// TIA Portal V19 program export: 2 tag tables, 1 data types, 4 data blocks, 27 code blocks (in call order from the OBs), 31 instance data blocks

VAR_GLOBAL   // PLC tag table "Default tag table"
   B0 AT %QB0 : Byte;
   B1 AT %QB1 : Byte;
   Clock_Byte AT %MB0 : Byte;
   Clock_10Hz AT %M0.0 : Bool;
   Clock_5Hz AT %M0.1 : Bool;
   "Clock_2.5Hz" AT %M0.2 : Bool;
   Clock_2Hz AT %M0.3 : Bool;
   "Clock_1.25Hz" AT %M0.4 : Bool;
   Clock_1Hz AT %M0.5 : Bool;
   "Clock_0.625Hz" AT %M0.6 : Bool;
   "Clock_0.5Hz" AT %M0.7 : Bool;
   System_Byte AT %MB1 : Byte;
   FirstScan AT %M1.0 : Bool;
   DiagStatusUpdate AT %M1.1 : Bool;
   AlwaysTRUE AT %M1.2 : Bool;
   AlwaysFALSE AT %M1.3 : Bool;
   "from et200sp PLC_1" AT %IB100 : Byte;   // Clock Byte From ET200SP sent Left Coupler for Display on RIO 1
   toET200spfromPLC1 AT %QB100 : Byte;   // Clock Byte To ET200SP sent Left Coupler
   "from et200sp PLC_1 Right" AT %IB200 : Byte;   // Clock Byte From ET200SP sent Right Coupler for Display on RIO 1
   "toET200spfromPLC1 Right" AT %QB200 : Byte;   // Clock Byte To ET200SP sent Right Coupler
END_VAR

VAR_GLOBAL   // PLC tag table "LAcycCom_Common"
END_VAR
VAR_GLOBAL CONSTANT   // user constants
   LACYCCOM_BUFFER_ELEMENTS_UPPER_LIM : Int := 59;   // Upper limit of request buffer array
END_VAR

TYPE "NetworkSwitchHMI"
   STRUCT
      Ports { S7_SetPoint := 'True'} : Array[1..8] of "LPNDR_typePortInformation";
      Port { S7_SetPoint := 'True'} : "LPNDR_typePortInformation";
      Index { S7_SetPoint := 'True'} : Int := 1;
   END_STRUCT;
END_TYPE

DATA_BLOCK "GlobalDB"   // DB9
{ S7_Optimized_Access := 'FALSE' }
   VAR RETAIN
      RTInfo : Struct   // Used to collect runtime information on an individual FB/FC
         Mode : UInt := 1;
         OBnumber : OB_ANY := 1;
         Info_LTIME : LTime := LT#0NS;
         RetVal : Int := 0;
      END_STRUCT;
      Runtime : Struct   // Used to collect individual runtime information of OB
         OB1Scan : Struct
            Min : LReal := 1000.0;
            Max : LReal;
            Current { ExternalAccessible := 'False'; ExternalVisible := 'False'; ExternalWritable := 'False'} : LReal;
            temp { ExternalAccessible := 'False'; ExternalVisible := 'False'; ExternalWritable := 'False'} : LReal;
            Mem { ExternalAccessible := 'False'; ExternalVisible := 'False'; ExternalWritable := 'False'} : LReal := 0.0;
            PreviousScan { ExternalAccessible := 'False'; ExternalVisible := 'False'; ExternalWritable := 'False'} : LReal;
            ResetMin : Bool;
            "Reset Max" : Bool;
         END_STRUCT;
      END_STRUCT;
      Trigger_StopSynch : Struct   // Used to trigger the Swapping of Status on the Reundant PLC
         REQ_FullSwapSequence { S7_SetPoint := 'True'} : Bool;   // Trigger used to perform a full swap of PLCs
         REQ_StopPrimary { S7_SetPoint := 'True'} : Bool;   // trigger a primary stop
         REQ_SynchUp { S7_SetPoint := 'True'} : Bool;   // trigger a synchronization
         Mode_StopPrimary : Int := 8;   // Stop Primary = 8
         Mode_SynchUp : Int := 7;   // Synchronization = 7
         StopPrimary_Retry_Busy : Bool;   // triggered due to RHCTRL being busy
         SynchUp_Retry_Busy : Bool;   // triggered due to RHCTRL being busy
         SyncSequenceFlag : Bool;
         RH_CTRL_PrimaryStop : Struct   // Used to stop and synch primary or backup
            REQ : Bool;
            Ret_Val : Byte;
            Busy : Bool;
         END_STRUCT;
         RH_CTRL_SyncUp : Struct   // Used to stop and synch primary or backup
            REQ : Bool;
            Ret_Val : Byte;
            Busy : Bool;
         END_STRUCT;
         SyncSequenceTimer : IEC_TIMER;
         SequenceTimer : IEC_TIMER;   // Timer to sequence between stop and synch
         SequenceAlarm { S7_SetPoint := 'True'} : Bool;
      END_STRUCT;
      Network { S7_SetPoint := 'True'} : "NetworkSwitchHMI";   // Used to collect switch XC208 details
      SystemTime { S7_SetPoint := 'True'} : DTL;   // Used to record cycle time of code
      tempSystemTime { S7_SetPoint := 'True'} : Int;
      "Array" : Array[0..1000] of "typeDiagnostics";   // Test Array
   END_VAR
BEGIN
   Trigger_StopSynch.SequenceTimer.PT := T#25s;   // Time based on full sequence elapsed timer
END_DATA_BLOCK

DATA_BLOCK "DB_HMI Support"   // DB10000
{ S7_Optimized_Access := 'FALSE' }
// stored: AutoNumber false
   VAR
      "PLC Mode" : Int;
      "PLC Near Status" : Int;
      "PLC Far Status" : Int;
      "Bypasses Status" : Int;
      OperationStateSystem : Int;
      MRPRingState : Int;
   END_VAR
BEGIN
END_DATA_BLOCK

DATA_BLOCK "hmiDatatransferTP1200"   // DB10
{ S7_Optimized_Access := 'TRUE' }
// stored: AutoNumber false, MemoryReserve 100
   VAR
      plc1LedState : Int;
      plc2LedState : Int;
      plcOperationState : Int;
      plcMrpState : Int;
      plcStopMonitoring : Int;
   END_VAR
BEGIN
END_DATA_BLOCK

DATA_BLOCK "EnS_Buffer32469"   // DB2
TITLE = Global DB for buffer data
AUTHOR : Siemens
FAMILY : EnS
// Global DB for buffer data
   STRUCT
      EnS_Buffer32469 : Array[0..114] of "EnS_typeValue";
   END_STRUCT;
BEGIN
END_DATA_BLOCK

ORGANIZATION_BLOCK "Main"   // OB1, LAD, ProgramCycle
TITLE = "Main Program Sweep (Cycle)"
{ S7_Optimized_Access := 'TRUE' }
// stored: AutoNumber false, SetENOAutomatically false
   VAR_INPUT
      Initial_Call : Bool;   // Initial call of this OB
      Remanence : Bool;   // =True, if remanent data are available
   END_VAR
BEGIN

REGION Network 1: Map clock byte to output of dq card
   // Display "to" and "from" using move command for troubleshooting
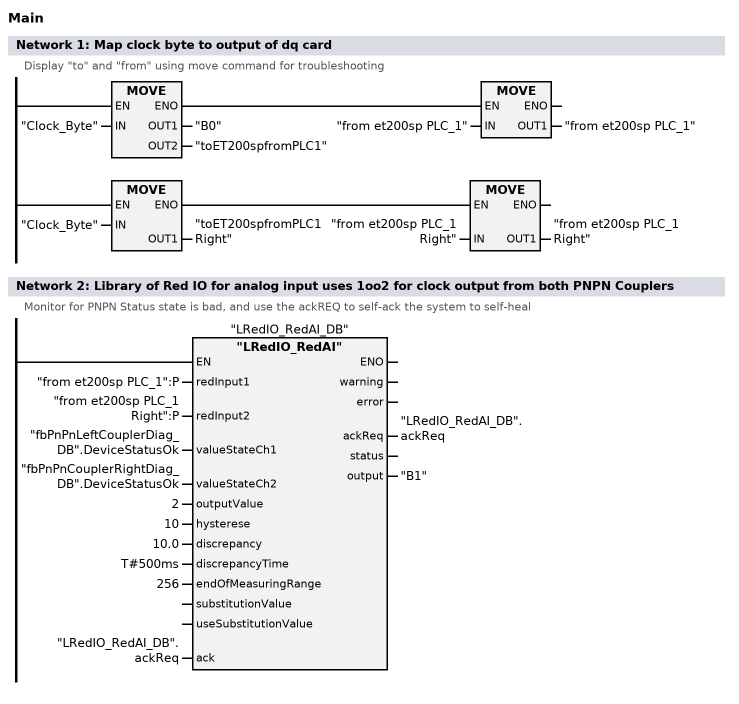
   RUNG wire#powerrail
      Move(in := "Clock_Byte", out1 => "B0", out2 => "toET200spfromPLC1")
      Move(in := "from et200sp PLC_1", out1 => "from et200sp PLC_1")
   END_RUNG
   RUNG wire#powerrail
      Move(in := "Clock_Byte", out1 => "toET200spfromPLC1 Right")
      Move(in := "from et200sp PLC_1 Right", out1 => "from et200sp PLC_1 Right")
   END_RUNG
   // the same network as SCL:
   "B0" := "Clock_Byte";
   "toET200spfromPLC1" := "Clock_Byte";
   "from et200sp PLC_1" := "from et200sp PLC_1";
   "toET200spfromPLC1 Right" := "Clock_Byte";
   "from et200sp PLC_1 Right" := "from et200sp PLC_1 Right";
END_REGION

REGION Network 2: Library of Red IO for analog input uses 1oo2 for clock output from both PNPN Couplers
   // Monitor for PNPN Status state is bad, and use the ackREQ to self-ack the system to self-heal
   RUNG wire#powerrail
      "LRedIO_RedAI_DB"(redInput1 := "from et200sp PLC_1":P, redInput2 := "from et200sp PLC_1 Right":P, valueStateCh1 := "fbPnPnLeftCouplerDiag_DB".DeviceStatusOk, valueStateCh2 := "fbPnPnCouplerRightDiag_DB".DeviceStatusOk, outputValue := 2, hysterese := 10, discrepancy := 10.0, discrepancyTime := T#500ms, endOfMeasuringRange := 256, substitutionValue :=, useSubstitutionValue :=, ack := "LRedIO_RedAI_DB".ackReq, warning =>, error =>, ackReq => "LRedIO_RedAI_DB".ackReq, status =>, output => "B1")
   END_RUNG
   // the same network as SCL:
   "LRedIO_RedAI_DB"(redInput1 := "from et200sp PLC_1":P,   // "LRedIO_RedAI"
                     redInput2 := "from et200sp PLC_1 Right":P,
                     valueStateCh1 := "fbPnPnLeftCouplerDiag_DB".DeviceStatusOk,
                     valueStateCh2 := "fbPnPnCouplerRightDiag_DB".DeviceStatusOk,
                     outputValue := 2,
                     hysterese := 10,
                     discrepancy := 10.0,
                     discrepancyTime := T#500ms,
                     endOfMeasuringRange := 256,
                     ack := "LRedIO_RedAI_DB".ackReq,
                     ackReq => "LRedIO_RedAI_DB".ackReq,
                     output => "B1");
END_REGION
END_ORGANIZATION_BLOCK

ORGANIZATION_BLOCK "RT_Info_Cyclic"   // OB30, LAD, CyclicInterrupt
{ S7_Optimized_Access := 'TRUE' }
// stored: SetENOAutomatically false
   VAR_INPUT
      Initial_Call : Bool;   // Initial call of this OB
      Event_Count : Int;   // Events discarded
   END_VAR
   VAR CONSTANT
      constRunSoloState : Int := 37;
      constRunRedundant : Int := 40;
   END_VAR
   VAR_TEMP   // added for the SCL form of the ladder/FBD networks
      _w1 : Bool;
      _w2 : Bool;
      _w3 : Bool;
      _w4 : Bool;
   END_VAR
BEGIN

REGION Network 1: RT_Info for specific OB
   // Used to find the specific runtime of an OB, change the OB number and see the INFO.
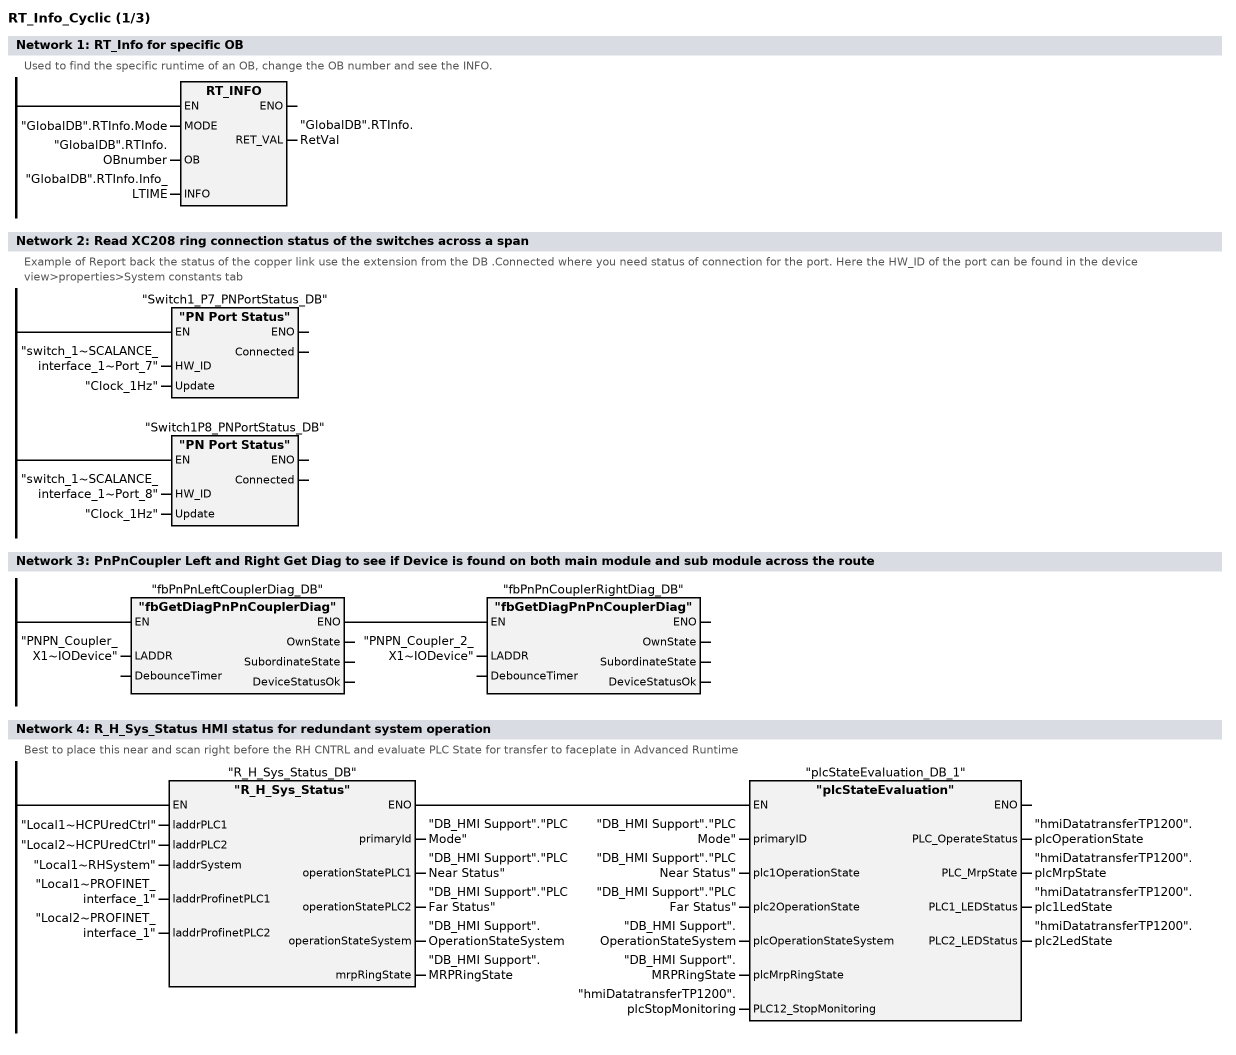
   RUNG wire#powerrail
      RT_INFO(MODE := "GlobalDB".RTInfo.Mode, OB := "GlobalDB".RTInfo.OBnumber, INFO := "GlobalDB".RTInfo.Info_LTIME, Ret_Val => "GlobalDB".RTInfo.RetVal)
   END_RUNG
   // the same network as SCL:
   "GlobalDB".RTInfo.RetVal := RT_INFO(MODE := "GlobalDB".RTInfo.Mode,
                           OB := "GlobalDB".RTInfo.OBnumber,
                           INFO := "GlobalDB".RTInfo.Info_LTIME);
END_REGION

REGION Network 2: Read XC208 ring connection status of the switches across a span
   // Example of Report back the status of the copper link use the extension from the DB .Connected where you need status of connection for the port. Here the HW_ID of the port can be found in the device view>properties>System constants tab
   RUNG wire#powerrail
      "Switch1_P7_PNPortStatus_DB"(HW_ID := "switch_1~SCALANCE_interface_1~Port_7", Update := "Clock_1Hz", Connected =>)
   END_RUNG
   RUNG wire#powerrail
      "Switch1P8_PNPortStatus_DB"(HW_ID := "switch_1~SCALANCE_interface_1~Port_8", Update := "Clock_1Hz", Connected =>)
   END_RUNG
   // the same network as SCL:
   "Switch1_P7_PNPortStatus_DB"(HW_ID := "switch_1~SCALANCE_interface_1~Port_7", Update := "Clock_1Hz");   // "PN Port Status"
   "Switch1P8_PNPortStatus_DB"(HW_ID := "switch_1~SCALANCE_interface_1~Port_8", Update := "Clock_1Hz");   // "PN Port Status"
END_REGION

REGION Network 3: PnPnCoupler Left and Right Get Diag to see if Device is found on both main module and sub module across the route
   RUNG wire#powerrail
      "fbPnPnLeftCouplerDiag_DB"(LADDR := "PNPN_Coupler_X1~IODevice", DebounceTimer :=, OwnState =>, SubordinateState =>, DeviceStatusOk =>)
      "fbPnPnCouplerRightDiag_DB"(LADDR := "PNPN_Coupler_2_X1~IODevice", DebounceTimer :=, OwnState =>, SubordinateState =>, DeviceStatusOk =>)
   END_RUNG
   // the same network as SCL:
   "fbPnPnLeftCouplerDiag_DB"(LADDR := "PNPN_Coupler_X1~IODevice", ENO => #_w1);   // "fbGetDiagPnPnCouplerDiag"
   IF #_w1 THEN
       "fbPnPnCouplerRightDiag_DB"(LADDR := "PNPN_Coupler_2_X1~IODevice");   // "fbGetDiagPnPnCouplerDiag"
   END_IF;
END_REGION

REGION Network 4: R_H_Sys_Status HMI status for redundant system operation
   // Best to place this near and scan right before the RH CNTRL and evaluate PLC State for transfer to faceplate in Advanced Runtime
   RUNG wire#powerrail
      "R_H_Sys_Status_DB"(laddrPLC1 := "Local1~HCPUredCtrl", laddrPLC2 := "Local2~HCPUredCtrl", laddrSystem := "Local1~RHSystem", laddrProfinetPLC1 := "Local1~PROFINET_interface_1", laddrProfinetPLC2 := "Local2~PROFINET_interface_1", primaryId => "DB_HMI Support"."PLC Mode", operationStatePLC1 => "DB_HMI Support"."PLC Near Status", operationStatePLC2 => "DB_HMI Support"."PLC Far Status", operationStateSystem => "DB_HMI Support".OperationStateSystem, mrpRingState => "DB_HMI Support".MRPRingState)
      "plcStateEvaluation_DB_1"(primaryID := "DB_HMI Support"."PLC Mode", plc1OperationState := "DB_HMI Support"."PLC Near Status", plc2OperationState := "DB_HMI Support"."PLC Far Status", plcOperationStateSystem := "DB_HMI Support".OperationStateSystem, plcMrpRingState := "DB_HMI Support".MRPRingState, PLC12_StopMonitoring := "hmiDatatransferTP1200".plcStopMonitoring, PLC_OperateStatus => "hmiDatatransferTP1200".plcOperationState, PLC_MrpState => "hmiDatatransferTP1200".plcMrpState, PLC1_LEDStatus => "hmiDatatransferTP1200".plc1LedState, PLC2_LEDStatus => "hmiDatatransferTP1200".plc2LedState)
   END_RUNG
   // the same network as SCL:
   "R_H_Sys_Status_DB"(laddrPLC1 := "Local1~HCPUredCtrl",   // "R_H_Sys_Status"
                       laddrPLC2 := "Local2~HCPUredCtrl",
                       laddrSystem := "Local1~RHSystem",
                       laddrProfinetPLC1 := "Local1~PROFINET_interface_1",
                       laddrProfinetPLC2 := "Local2~PROFINET_interface_1",
                       primaryId => "DB_HMI Support"."PLC Mode",
                       operationStatePLC1 => "DB_HMI Support"."PLC Near Status",
                       operationStatePLC2 => "DB_HMI Support"."PLC Far Status",
                       operationStateSystem => "DB_HMI Support".OperationStateSystem,
                       mrpRingState => "DB_HMI Support".MRPRingState,
                       ENO => #_w1);
   IF #_w1 THEN
       "plcStateEvaluation_DB_1"(primaryID := "DB_HMI Support"."PLC Mode",   // "plcStateEvaluation"
                               plc1OperationState := "DB_HMI Support"."PLC Near Status",
                               plc2OperationState := "DB_HMI Support"."PLC Far Status",
                               plcOperationStateSystem := "DB_HMI Support".OperationStateSystem,
                               plcMrpRingState := "DB_HMI Support".MRPRingState,
                               PLC12_StopMonitoring := "hmiDatatransferTP1200".plcStopMonitoring,
                               PLC_OperateStatus => "hmiDatatransferTP1200".plcOperationState,
                               PLC_MrpState => "hmiDatatransferTP1200".plcMrpState,
                               PLC1_LEDStatus => "hmiDatatransferTP1200".plc1LedState,
                               PLC2_LEDStatus => "hmiDatatransferTP1200".plc2LedState);
   END_IF;
END_REGION

REGION Network 5: Trigger primary stop RH_CNTRL
   // Self Latching Sequence using FullSwap Sequence tag, independent function with REQ tag
   // Used to trigger Primary Stop based on input from stop primary and full swap boolean tag;
   //  positive edge triggered instruction RH_CTRL below.
   // This network uses a Primary stop request, and evaluates if the RH_CTRL is busy before 
   // changing the mode or moving on to the next step.
   // The Retry_Busy tag is used to record if a Busy bit was in place while being triggered to prevent moving
   //  mode during middle of RH_CTRL operation.
   // 
   // Modes:
   // 3: Disable execution of the SYNCUP
   // 4: Re-enable execution of the SYNCUP
   // 7: Request SYNCUP system state 
   // 8: Request STOP of the primary CPU
   // 9: Request STOP of the backup CPU
   // 
   // Use mode 8 to stop the primary PLC, then use Mode 7 to Synch the primary and backup.
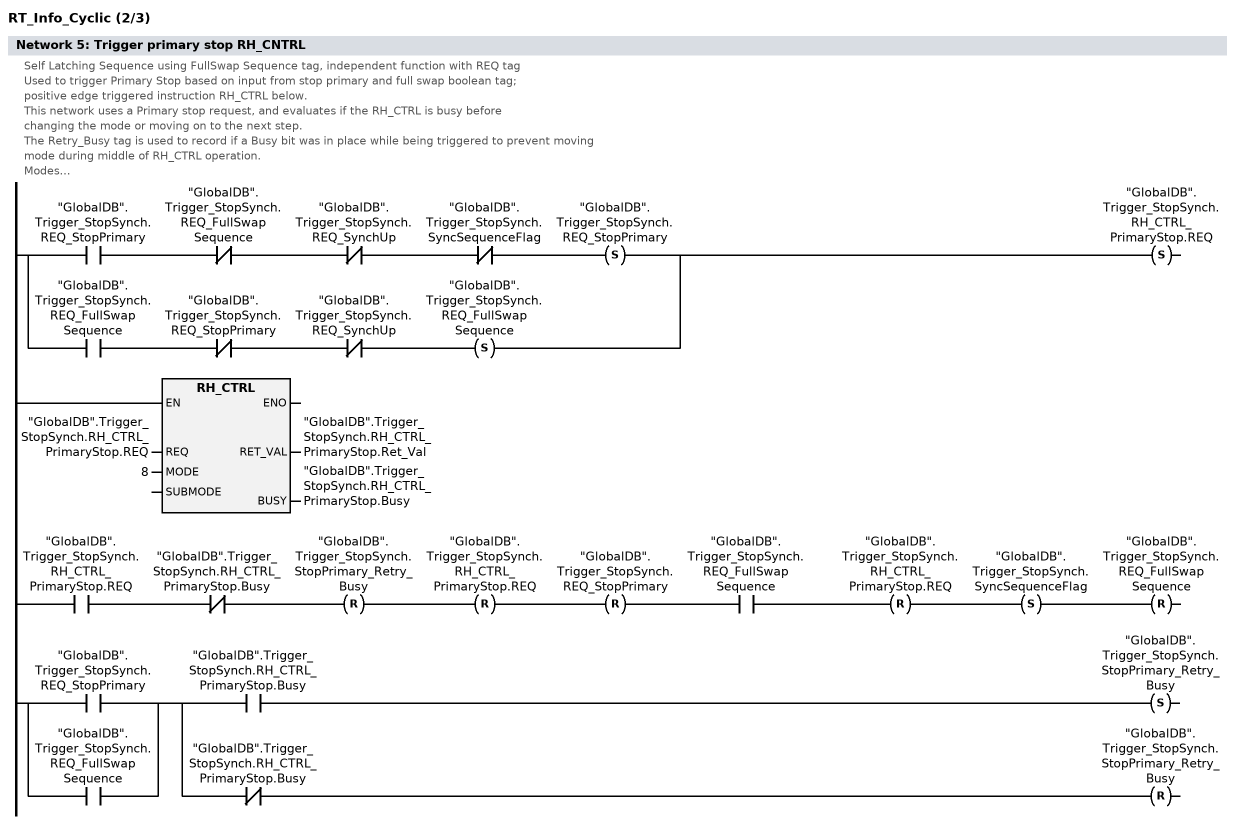
   RUNG wire#powerrail
      Contact( "GlobalDB".Trigger_StopSynch.REQ_StopPrimary )
      I_Contact( "GlobalDB".Trigger_StopSynch.REQ_FullSwapSequence )
      I_Contact( "GlobalDB".Trigger_StopSynch.REQ_SynchUp )
      I_Contact( "GlobalDB".Trigger_StopSynch.SyncSequenceFlag )
      S_Coil( "GlobalDB".Trigger_StopSynch.REQ_StopPrimary )
      wire#w1
      S_Coil( "GlobalDB".Trigger_StopSynch.RH_CTRL_PrimaryStop.REQ )
   END_RUNG
   RUNG wire#powerrail
      Contact( "GlobalDB".Trigger_StopSynch.REQ_FullSwapSequence )
      I_Contact( "GlobalDB".Trigger_StopSynch.REQ_StopPrimary )
      I_Contact( "GlobalDB".Trigger_StopSynch.REQ_SynchUp )
      S_Coil( "GlobalDB".Trigger_StopSynch.REQ_FullSwapSequence )
   END_RUNG wire#w1
   RUNG wire#powerrail
      RH_CTRL(REQ := "GlobalDB".Trigger_StopSynch.RH_CTRL_PrimaryStop.REQ, Mode := 8, Submode :=, Ret_Val => "GlobalDB".Trigger_StopSynch.RH_CTRL_PrimaryStop.Ret_Val, Busy => "GlobalDB".Trigger_StopSynch.RH_CTRL_PrimaryStop.Busy)
   END_RUNG
   RUNG wire#powerrail
      Contact( "GlobalDB".Trigger_StopSynch.RH_CTRL_PrimaryStop.REQ )
      I_Contact( "GlobalDB".Trigger_StopSynch.RH_CTRL_PrimaryStop.Busy )
      R_Coil( "GlobalDB".Trigger_StopSynch.StopPrimary_Retry_Busy )
      R_Coil( "GlobalDB".Trigger_StopSynch.RH_CTRL_PrimaryStop.REQ )
      R_Coil( "GlobalDB".Trigger_StopSynch.REQ_StopPrimary )
      Contact( "GlobalDB".Trigger_StopSynch.REQ_FullSwapSequence )
      R_Coil( "GlobalDB".Trigger_StopSynch.RH_CTRL_PrimaryStop.REQ )
      S_Coil( "GlobalDB".Trigger_StopSynch.SyncSequenceFlag )
      R_Coil( "GlobalDB".Trigger_StopSynch.REQ_FullSwapSequence )
   END_RUNG
   RUNG wire#powerrail
      Contact( "GlobalDB".Trigger_StopSynch.REQ_StopPrimary )
      wire#w2
      Contact( "GlobalDB".Trigger_StopSynch.RH_CTRL_PrimaryStop.Busy )
      S_Coil( "GlobalDB".Trigger_StopSynch.StopPrimary_Retry_Busy )
   END_RUNG
   RUNG wire#powerrail
      Contact( "GlobalDB".Trigger_StopSynch.REQ_FullSwapSequence )
   END_RUNG wire#w2
   RUNG wire#w2
      I_Contact( "GlobalDB".Trigger_StopSynch.RH_CTRL_PrimaryStop.Busy )
      R_Coil( "GlobalDB".Trigger_StopSynch.StopPrimary_Retry_Busy )
   END_RUNG
   // the same network as SCL:
   #_w1 := "GlobalDB".Trigger_StopSynch.REQ_StopPrimary AND NOT "GlobalDB".Trigger_StopSynch.REQ_FullSwapSequence AND NOT "GlobalDB".Trigger_StopSynch.REQ_SynchUp AND NOT "GlobalDB".Trigger_StopSynch.SyncSequenceFlag;
   IF #_w1 THEN "GlobalDB".Trigger_StopSynch.REQ_StopPrimary := TRUE; END_IF;
   #_w2 := "GlobalDB".Trigger_StopSynch.REQ_FullSwapSequence AND NOT "GlobalDB".Trigger_StopSynch.REQ_StopPrimary AND NOT "GlobalDB".Trigger_StopSynch.REQ_SynchUp;
   IF #_w2 THEN "GlobalDB".Trigger_StopSynch.REQ_FullSwapSequence := TRUE; END_IF;
   IF #_w1 OR #_w2 THEN "GlobalDB".Trigger_StopSynch.RH_CTRL_PrimaryStop.REQ := TRUE; END_IF;
   "GlobalDB".Trigger_StopSynch.RH_CTRL_PrimaryStop.Ret_Val := RH_CTRL(REQ := "GlobalDB".Trigger_StopSynch.RH_CTRL_PrimaryStop.REQ,
                           Mode := 8,
                           Busy => "GlobalDB".Trigger_StopSynch.RH_CTRL_PrimaryStop.Busy);
   #_w3 := "GlobalDB".Trigger_StopSynch.RH_CTRL_PrimaryStop.REQ AND NOT "GlobalDB".Trigger_StopSynch.RH_CTRL_PrimaryStop.Busy;
   IF #_w3 THEN
       "GlobalDB".Trigger_StopSynch.StopPrimary_Retry_Busy := FALSE;
       "GlobalDB".Trigger_StopSynch.RH_CTRL_PrimaryStop.REQ := FALSE;
       "GlobalDB".Trigger_StopSynch.REQ_StopPrimary := FALSE;
   END_IF;
   IF #_w3 AND "GlobalDB".Trigger_StopSynch.REQ_FullSwapSequence THEN
       "GlobalDB".Trigger_StopSynch.RH_CTRL_PrimaryStop.REQ := FALSE;
       "GlobalDB".Trigger_StopSynch.SyncSequenceFlag := TRUE;
       "GlobalDB".Trigger_StopSynch.REQ_FullSwapSequence := FALSE;
   END_IF;
   #_w4 := "GlobalDB".Trigger_StopSynch.REQ_StopPrimary OR "GlobalDB".Trigger_StopSynch.REQ_FullSwapSequence;
   IF #_w4 AND "GlobalDB".Trigger_StopSynch.RH_CTRL_PrimaryStop.Busy THEN
       "GlobalDB".Trigger_StopSynch.StopPrimary_Retry_Busy := TRUE;
   END_IF;
   IF #_w4 AND NOT "GlobalDB".Trigger_StopSynch.RH_CTRL_PrimaryStop.Busy THEN
       "GlobalDB".Trigger_StopSynch.StopPrimary_Retry_Busy := FALSE;
   END_IF;
END_REGION

REGION Network 6: Trigger Synch up RH_CNTRL
   // Self Latching Sequence using FullSwap Sequence tag, independent function with REQ tag
   // Used to trigger Sync up; positive edge triggered instruction RH_CTRL below
   // Sequence can also be triggered by Full sequence request which can set the SyncSequenceFlag below
   // SyncSequence Flag is help for next step until run Run-Solo status is reported
   //  positive edge triggered instruction RH_CTRL below
   // This network uses a synch up request, and evaluates if the RH_CTRL is busy before changing the mode
   // The Retry_Busy tag is used to record if a Busy bit was in place while being triggered to prevent moving
   //  mode during middle of RH_CTRL operation
   // 
   // Modes:
   // 3: Disable execution of the SYNCUP
   // 4: Re-enable execution of the SYNCUP
   // 7: Request SYNCUP system state 
   // 8: Request STOP of the primary CPU
   // 9: Request STOP of the backup CPU
   // 
   // Use mode 8 to stop the primary PLC, then use Mode 7 to Synch the primary and backup.
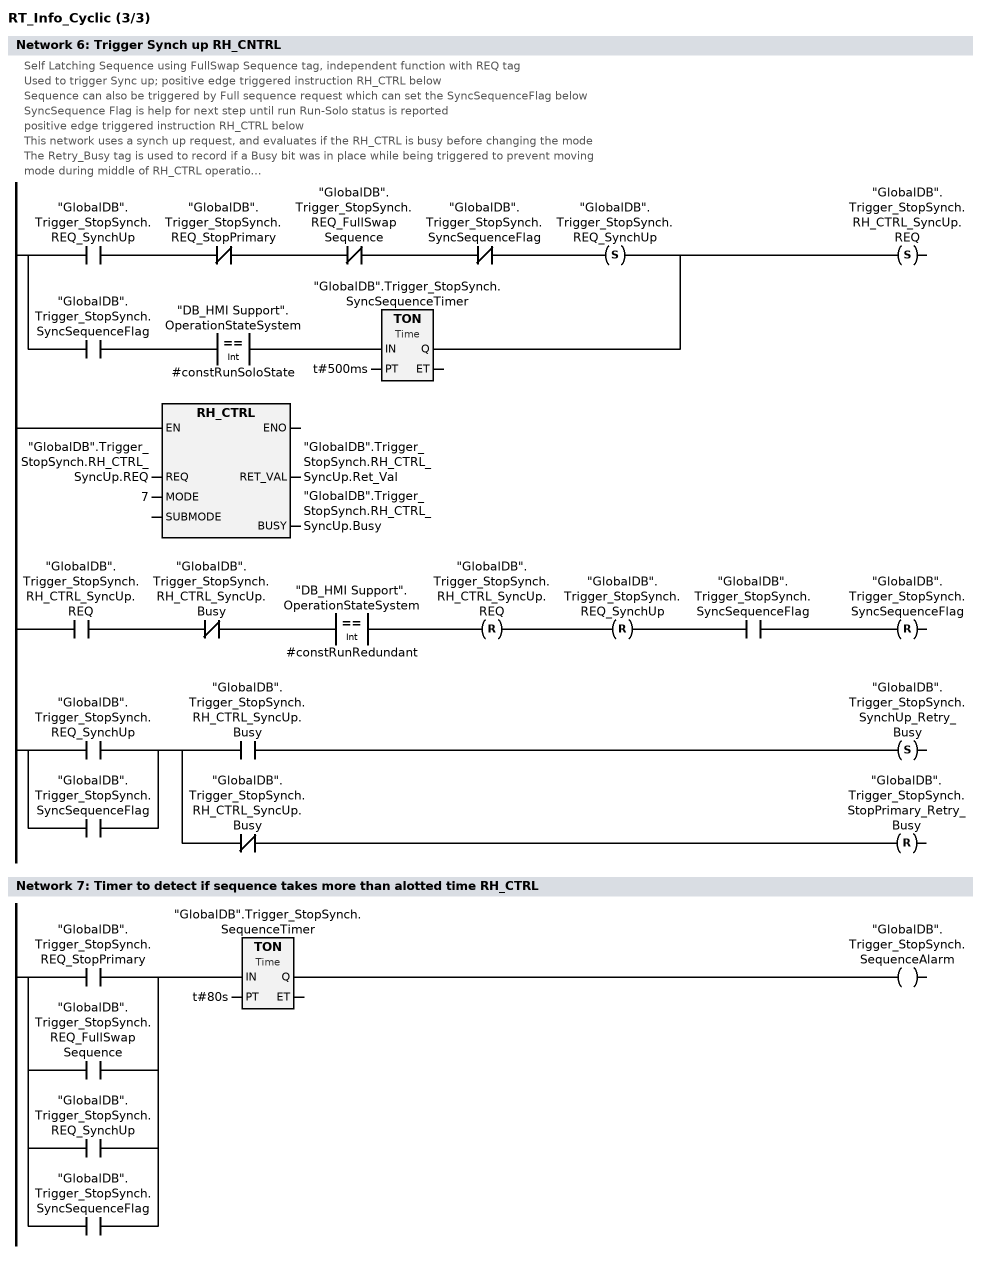
   RUNG wire#powerrail
      Contact( "GlobalDB".Trigger_StopSynch.REQ_SynchUp )
      I_Contact( "GlobalDB".Trigger_StopSynch.REQ_StopPrimary )
      I_Contact( "GlobalDB".Trigger_StopSynch.REQ_FullSwapSequence )
      I_Contact( "GlobalDB".Trigger_StopSynch.SyncSequenceFlag )
      S_Coil( "GlobalDB".Trigger_StopSynch.REQ_SynchUp )
      wire#w1
      S_Coil( "GlobalDB".Trigger_StopSynch.RH_CTRL_SyncUp.REQ )
   END_RUNG
   RUNG wire#powerrail
      Contact( "GlobalDB".Trigger_StopSynch.SyncSequenceFlag )
      { S7_Templates := "SrcType := Int" } EQ_Contact(in1 := "DB_HMI Support".OperationStateSystem, in2 := #constRunSoloState)
      { S7_Templates := "time_type := Time" } "GlobalDB".Trigger_StopSynch.SyncSequenceTimer.TON(pt := t#500ms, et =>)
   END_RUNG wire#w1
   RUNG wire#powerrail
      RH_CTRL(REQ := "GlobalDB".Trigger_StopSynch.RH_CTRL_SyncUp.REQ, Mode := 7, Submode :=, Ret_Val => "GlobalDB".Trigger_StopSynch.RH_CTRL_SyncUp.Ret_Val, Busy => "GlobalDB".Trigger_StopSynch.RH_CTRL_SyncUp.Busy)
   END_RUNG
   RUNG wire#powerrail
      Contact( "GlobalDB".Trigger_StopSynch.RH_CTRL_SyncUp.REQ )
      I_Contact( "GlobalDB".Trigger_StopSynch.RH_CTRL_SyncUp.Busy )
      { S7_Templates := "SrcType := Int" } EQ_Contact(in1 := "DB_HMI Support".OperationStateSystem, in2 := #constRunRedundant)
      R_Coil( "GlobalDB".Trigger_StopSynch.RH_CTRL_SyncUp.REQ )
      R_Coil( "GlobalDB".Trigger_StopSynch.REQ_SynchUp )
      Contact( "GlobalDB".Trigger_StopSynch.SyncSequenceFlag )
      R_Coil( "GlobalDB".Trigger_StopSynch.SyncSequenceFlag )
   END_RUNG
   RUNG wire#powerrail
      Contact( "GlobalDB".Trigger_StopSynch.REQ_SynchUp )
      wire#w2
      Contact( "GlobalDB".Trigger_StopSynch.RH_CTRL_SyncUp.Busy )
      S_Coil( "GlobalDB".Trigger_StopSynch.SynchUp_Retry_Busy )
   END_RUNG
   RUNG wire#powerrail
      Contact( "GlobalDB".Trigger_StopSynch.SyncSequenceFlag )
   END_RUNG wire#w2
   RUNG wire#w2
      I_Contact( "GlobalDB".Trigger_StopSynch.RH_CTRL_SyncUp.Busy )
      R_Coil( "GlobalDB".Trigger_StopSynch.StopPrimary_Retry_Busy )
   END_RUNG
   // the same network as SCL:
   #_w1 := "GlobalDB".Trigger_StopSynch.REQ_SynchUp AND NOT "GlobalDB".Trigger_StopSynch.REQ_StopPrimary AND NOT "GlobalDB".Trigger_StopSynch.REQ_FullSwapSequence AND NOT "GlobalDB".Trigger_StopSynch.SyncSequenceFlag;
   IF #_w1 THEN "GlobalDB".Trigger_StopSynch.REQ_SynchUp := TRUE; END_IF;
   "GlobalDB".Trigger_StopSynch.SyncSequenceTimer.TON(IN := "GlobalDB".Trigger_StopSynch.SyncSequenceFlag AND ("DB_HMI Support".OperationStateSystem = #constRunSoloState),
                           PT := t#500ms);
   IF #_w1 OR "GlobalDB".Trigger_StopSynch.SyncSequenceTimer.Q THEN
       "GlobalDB".Trigger_StopSynch.RH_CTRL_SyncUp.REQ := TRUE;
   END_IF;
   "GlobalDB".Trigger_StopSynch.RH_CTRL_SyncUp.Ret_Val := RH_CTRL(REQ := "GlobalDB".Trigger_StopSynch.RH_CTRL_SyncUp.REQ,
                           Mode := 7,
                           Busy => "GlobalDB".Trigger_StopSynch.RH_CTRL_SyncUp.Busy);
   #_w2 := "GlobalDB".Trigger_StopSynch.RH_CTRL_SyncUp.REQ AND NOT "GlobalDB".Trigger_StopSynch.RH_CTRL_SyncUp.Busy AND ("DB_HMI Support".OperationStateSystem = #constRunRedundant);
   IF #_w2 THEN
       "GlobalDB".Trigger_StopSynch.RH_CTRL_SyncUp.REQ := FALSE;
       "GlobalDB".Trigger_StopSynch.REQ_SynchUp := FALSE;
   END_IF;
   IF #_w2 AND "GlobalDB".Trigger_StopSynch.SyncSequenceFlag THEN
       "GlobalDB".Trigger_StopSynch.SyncSequenceFlag := FALSE;
   END_IF;
   #_w3 := "GlobalDB".Trigger_StopSynch.REQ_SynchUp OR "GlobalDB".Trigger_StopSynch.SyncSequenceFlag;
   IF #_w3 AND "GlobalDB".Trigger_StopSynch.RH_CTRL_SyncUp.Busy THEN
       "GlobalDB".Trigger_StopSynch.SynchUp_Retry_Busy := TRUE;
   END_IF;
   IF #_w3 AND NOT "GlobalDB".Trigger_StopSynch.RH_CTRL_SyncUp.Busy THEN
       "GlobalDB".Trigger_StopSynch.StopPrimary_Retry_Busy := FALSE;
   END_IF;
END_REGION

REGION Network 7: Timer to detect if sequence takes more than alotted time RH_CTRL
   RUNG wire#powerrail
      Contact( "GlobalDB".Trigger_StopSynch.REQ_StopPrimary )
      wire#w1
      { S7_Templates := "time_type := Time" } "GlobalDB".Trigger_StopSynch.SequenceTimer.TON(pt := t#80s, et =>)
      Coil( "GlobalDB".Trigger_StopSynch.SequenceAlarm )
   END_RUNG
   RUNG wire#powerrail
      Contact( "GlobalDB".Trigger_StopSynch.REQ_FullSwapSequence )
   END_RUNG wire#w1
   RUNG wire#powerrail
      Contact( "GlobalDB".Trigger_StopSynch.REQ_SynchUp )
   END_RUNG wire#w1
   RUNG wire#powerrail
      Contact( "GlobalDB".Trigger_StopSynch.SyncSequenceFlag )
   END_RUNG wire#w1
   // the same network as SCL:
   "GlobalDB".Trigger_StopSynch.SequenceTimer.TON(IN := "GlobalDB".Trigger_StopSynch.REQ_StopPrimary OR "GlobalDB".Trigger_StopSynch.REQ_FullSwapSequence OR "GlobalDB".Trigger_StopSynch.REQ_SynchUp OR "GlobalDB".Trigger_StopSynch.SyncSequenceFlag,
                           PT := t#80s);
   "GlobalDB".Trigger_StopSynch.SequenceAlarm := "GlobalDB".Trigger_StopSynch.SequenceTimer.Q;
END_REGION
END_ORGANIZATION_BLOCK

FUNCTION_BLOCK "PN Port Status"   // FB5, LAD
{ S7_Optimized_Access := 'TRUE' }
// stored: MemoryReserve 100, SetENOAutomatically false
   VAR_INPUT
      HW_ID : HW_IO;
      Update : Bool;
   END_VAR
   VAR_OUTPUT
      Connected : Bool;
   END_VAR
   VAR
      Updated_ReqP : Bool;
      Updated_Req : Bool;
      RDREC_Instance { S7_SetPoint := 'True'} : RDREC;
   END_VAR
   VAR_TEMP
      Record : Struct
         BlockType : Word;
         BlockLength : UInt;
         BlockVersionHigh : USInt;
         BlockVersionLow : USInt;
         Padding : Word;
         SlotNumber : Word;
         SubSlotNumber : Word;
         Data : Array[0..299] of Byte;
      END_STRUCT;
      n : Array[0..3] of UInt;
      LinkState : Word;
   END_VAR
   VAR_TEMP   // added for the SCL form of the ladder/FBD networks
      _w1 : Bool;
   END_VAR
BEGIN

REGION Network 1: Positive Edge triggered Update Req
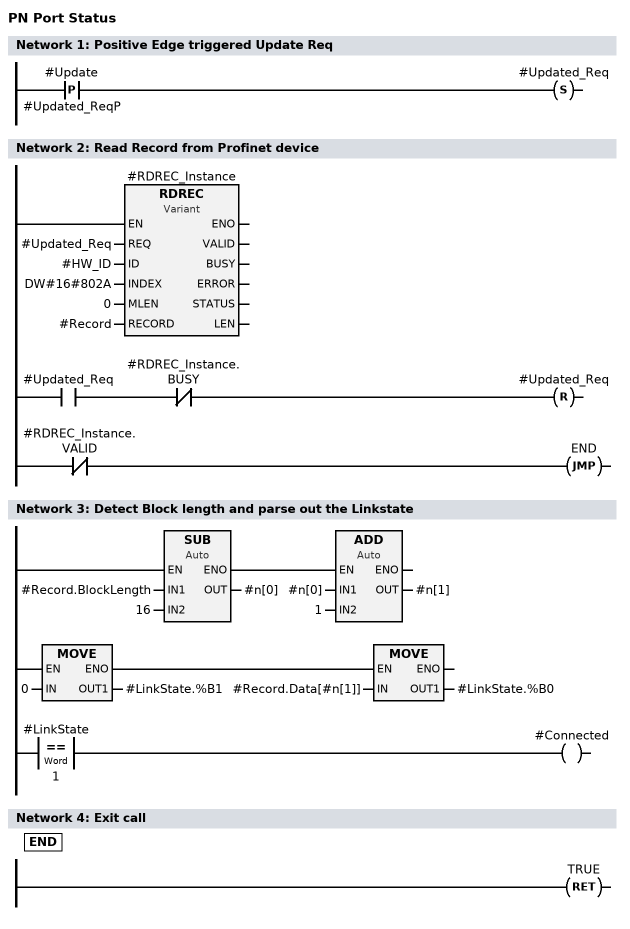
   RUNG wire#powerrail
      P_Contact(operand := #Update, bit := #Updated_ReqP)
      S_Coil( #Updated_Req )
   END_RUNG
   // the same network as SCL:
   #_w1 := #Update AND NOT #Updated_ReqP;   // rising edge of #Update
   #Updated_ReqP := #Update;
   IF #_w1 THEN #Updated_Req := TRUE; END_IF;
END_REGION

REGION Network 2: Read Record from Profinet device
   RUNG wire#powerrail
      { S7_Templates := "[ptr_type := Variant, id_type := HW_IO, index_type := DInt, len_type := UInt]" } #RDREC_Instance.RDREC(REQ := #Updated_Req, ID := #HW_ID, INDEX := DW#16#802A, MLEN := 0, RECORD := #Record, VALID =>, BUSY =>, ERROR =>, STATUS =>, LEN =>)
   END_RUNG
   RUNG wire#powerrail
      Contact( #Updated_Req )
      I_Contact( #RDREC_Instance.BUSY )
      R_Coil( #Updated_Req )
   END_RUNG
   RUNG wire#powerrail
      I_Contact( #RDREC_Instance.VALID )
      JumpCoil( END )
   END_RUNG
   // the same network as SCL:
   #RDREC_Instance(REQ := #Updated_Req, ID := #HW_ID, INDEX := DW#16#802A, MLEN := 0, RECORD := #Record);   // RDREC
   IF #Updated_Req AND NOT #RDREC_Instance.BUSY THEN #Updated_Req := FALSE; END_IF;
   IF NOT #RDREC_Instance.VALID THEN GOTO END; END_IF;
END_REGION

REGION Network 3: Detect Block length and parse out the Linkstate
   RUNG wire#powerrail
      Sub(in1 := #Record.BlockLength, in2 := 16, out => #n[0])
      Add(in1 := #n[0], in2 := 1, out => #n[1])
   END_RUNG
   RUNG wire#powerrail
      Move(in := 0, out1 => #LinkState.%B1)
      Move(in := #Record.Data[#n[1]], out1 => #LinkState.%B0)
   END_RUNG
   RUNG wire#powerrail
      { S7_Templates := "SrcType := Word" } EQ_Contact(in1 := #LinkState, in2 := 1)
      Coil( #Connected )
   END_RUNG
   // the same network as SCL:
   #n[0] := #Record.BlockLength - 16;
   #n[1] := #n[0] + 1;
   #LinkState.%B1 := 0;
   #LinkState.%B0 := #Record.Data[#n[1]];
   #Connected := #LinkState = 1;
END_REGION

REGION Network 4: Exit call
   END:
   ENO := TRUE;
   RETURN;
END_REGION
END_FUNCTION_BLOCK

FUNCTION_BLOCK "fbGetDiagPnPnCouplerDiag"   // FB1, LAD
{ S7_Optimized_Access := 'TRUE' }
// stored: MemoryReserve 100, SetENOAutomatically false
   VAR_INPUT
      LADDR : HW_ANY;   // Hardware Address of the ~IODevice number
      DebounceTimer : Time := T#3ms;
   END_VAR
   VAR_OUTPUT
      OwnState : UInt;
      SubordinateState : UInt;
      DeviceStatusOk : Bool;
   END_VAR
   VAR
      Diag : DIS;
      Sub { S7_SetPoint := 'True'} : DNN;
      RetValueDiag : Int;
      CntDiagDiag : UInt;
      RetValueSub : Int;
      CntDiagSub : UInt;
      BadStateDebounceTimer : IEC_TIMER;
   END_VAR
   VAR CONSTANT
      "IO Device Mode" : Int := 1;
      "Subordinate device Mode" : Int := 2;
   END_VAR
   VAR_TEMP   // added for the SCL form of the ladder/FBD networks
      _w1 : Bool;
   END_VAR
BEGIN

REGION Network 1: PnPnCoupler Left Get Diag
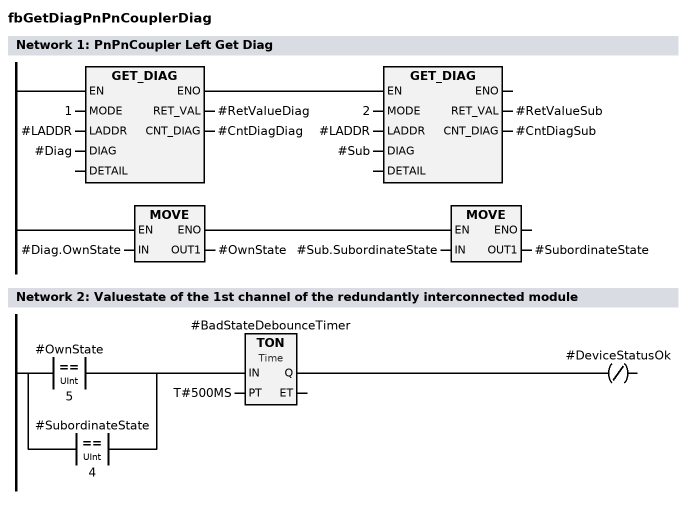
   RUNG wire#powerrail
      GET_DIAG(MODE := 1, LADDR := #LADDR, DIAG := #Diag, DETAIL :=, RET_VAL => #RetValueDiag, CNT_DIAG => #CntDiagDiag)
      GET_DIAG(MODE := 2, LADDR := #LADDR, DIAG := #Sub, DETAIL :=, RET_VAL => #RetValueSub, CNT_DIAG => #CntDiagSub)
   END_RUNG
   RUNG wire#powerrail
      Move(in := #Diag.OwnState, out1 => #OwnState)
      Move(in := #Sub.SubordinateState, out1 => #SubordinateState)
   END_RUNG
   // the same network as SCL:
   #RetValueDiag := GET_DIAG(MODE := 1, LADDR := #LADDR, DIAG := #Diag, CNT_DIAG => #CntDiagDiag, ENO => #_w1);
   IF #_w1 THEN
       #RetValueSub := GET_DIAG(MODE := 2, LADDR := #LADDR, DIAG := #Sub, CNT_DIAG => #CntDiagSub);
   END_IF;
   #OwnState := #Diag.OwnState;
   #SubordinateState := #Sub.SubordinateState;
END_REGION

REGION Network 2: Valuestate of the 1st channel of the redundantly interconnected module
   RUNG wire#powerrail
      { S7_Templates := "SrcType := UInt" } EQ_Contact(in1 := #OwnState, in2 := 5)
      wire#w1
      { S7_Templates := "time_type := Time" } #BadStateDebounceTimer.TON(pt := T#500MS, et =>)
      I_Coil( #DeviceStatusOk )
   END_RUNG
   RUNG wire#powerrail
      { S7_Templates := "SrcType := UInt" } EQ_Contact(in1 := #SubordinateState, in2 := 4)
   END_RUNG wire#w1
   // the same network as SCL:
   #BadStateDebounceTimer.TON(IN := (#OwnState = 5) OR (#SubordinateState = 4), PT := T#500MS);
   #DeviceStatusOk := NOT #BadStateDebounceTimer.Q;
END_REGION
END_FUNCTION_BLOCK

FUNCTION_BLOCK "R_H_Sys_Status"
{ S7_Optimized_Access := 'TRUE' }
VERSION : 0.1
   VAR_INPUT 
      laddrPLC1 : HW_ANY;
      laddrPLC2 : HW_ANY;
      laddrSystem : HW_ANY;
      laddrProfinetPLC1 : HW_ANY;
      laddrProfinetPLC2 : HW_ANY;
   END_VAR

   VAR_OUTPUT 
      primaryId : Int;
      operationStatePLC1 : UInt;
      operationStatePLC2 : UInt;
      operationStateSystem : UInt;
      mrpRingState : UInt;
   END_VAR

   VAR 
      statDiagModeCpu1 { S7_SetPoint := 'True'} : UInt := 1;
      statCountDiagDetailsCpu1 : UInt;
      statReturnValueCpu1 : Int;
      statDiagCpu1 {InstructionName := 'DIS'; LibVersion := '1.0'; ExternalAccessible := 'False'; ExternalVisible := 'False'; ExternalWritable := 'False'} : DIS;
      statDiagModeCpu2 { S7_SetPoint := 'True'} : UInt := 1;
      statCountDiagDetailsCpu2 : UInt;
      statReturnValueCpu2 : Int;
      statDiagCpu2 {InstructionName := 'DIS'; LibVersion := '1.0'; ExternalAccessible := 'False'; ExternalVisible := 'False'; ExternalWritable := 'False'} : DIS;
      statDiagModeSystem { S7_SetPoint := 'True'} : UInt := 1;
      statCountDiagDetailsSystem : UInt;
      statReturnValueSystem : Int;
      statDiagSystem {InstructionName := 'DIS'; LibVersion := '1.0'; ExternalAccessible := 'False'; ExternalVisible := 'False'; ExternalWritable := 'False'} : DIS;
      statDataRecord1 : "LPNDR_typeMrpInformation";
      statDataRecord2 : "LPNDR_typeMrpInformation";
      statLPNDR_ReadMrpState { S7_SetPoint := 'True'} : HW_ANY;
      statLPNDR_ReadGlobalInfo_DB1 : "LPNDR_ReadGlobalInfo";
      statLPNDR_ReadGlobalInfo_DB2 : "LPNDR_ReadGlobalInfo";
      statLPNDR_ReadMrpState_DB : "LPNDR_ReadMrpState";
      statExecuteClock : Bool;
      IEC_Timer_0_Instance {InstructionName := 'TOF_TIME'; LibVersion := '1.0'} : TOF_TIME;
      statToggleExecuteClock { S7_SetPoint := 'True'} : Bool;
      statUndefinedState : Bool;
      statExecuteClock2 : Bool;
      statToggleExecuteClock2 : Bool;
      IEC_Timer_0_Instance_1 {InstructionName := 'TOF_TIME'; LibVersion := '1.0'} : TOF_TIME;
      IEC_Timer_0_Instance_2 {InstructionName := 'TOF_TIME'; LibVersion := '1.0'} : TOF_TIME;
      statError1 : Bool;
      statChoose1 : Bool;
      IEC_Timer_0_Instance_3 {InstructionName := 'TOF_TIME'; LibVersion := '1.0'} : TOF_TIME;
      statError2 : Bool;
      statChoose2 : Bool;
   END_VAR

   VAR_TEMP 
      tempGblInfoBusy1 : Bool;
      tempGblInfoDone1 : Bool;
      tempGblInfoError1 : Bool;
      tempGblInfoStatus1 : Word;
      tempGblInfoBusy2 : Bool;
      tempGblInfoDone2 : Bool;
      tempGblInfoError2 : Bool;
      tempGblInfoStatus2 : Word;
      tempMrpBusy : Bool;
      tempMrpDone : Bool;
      tempMrpError : Bool;
      tempMrpStatus : Word;
   END_VAR


BEGIN
	//=============================================================================
	// Siemens// (c)Copyright (2019)
	//-----------------------------------------------------------------------------
	// Tested with: S7 - 1517H & S7 - 1515R
	// Engineering: TIA Portal (V15.1)
	// Restrictions: only with S7 - 1500R&H
	// Requirements: S7 - 1500R&H
	// Functionality: Diagnostics for S7 - 1500R & H systems for operating states, MRP-Ring and synchronisation state.
	//-----------------------------------------------------------------------------
	// Change log table:
	// Version Date Expert in charge Changes applied
	// 01.00.00 dd.mm.yyyy (Name of expert) First released version //=============================================================================
	//////////////////////////////////////////////////////////////////////////////////////////////////////////////////////////////////////////////
	
	// Check Primary CPU
	#primaryId := RH_GetPrimaryID();
	
	//Check Operationmode of CPU1 and CPU2 and System1 and System2
	#statReturnValueCpu1 := GET_DIAG(MODE := #statDiagModeCpu1, LADDR := #laddrPLC1, CNT_DIAG => #statCountDiagDetailsCpu1, DIAG := #statDiagCpu1);
	#statReturnValueCpu2 := GET_DIAG(MODE := #statDiagModeCpu2, LADDR := #laddrPLC2, CNT_DIAG => #statCountDiagDetailsCpu2, DIAG := #statDiagCpu2);
	#statReturnValueSystem := GET_DIAG(MODE := #statDiagModeSystem, LADDR := #laddrSystem, CNT_DIAG => #statCountDiagDetailsSystem, DIAG := #statDiagSystem);
	
	#operationStatePLC1 := #statDiagCpu1.OperatingState;
	#operationStatePLC2 := #statDiagCpu2.OperatingState;
	#operationStateSystem := #statDiagSystem.OperatingState;
	
	//Checking MRP - Ring
	#statLPNDR_ReadGlobalInfo_DB1(execute := #statExecuteClock,
	                              hwId := #laddrProfinetPLC1,
	                              mode := 2,
	                              busy => #tempGblInfoBusy1,
	                              done => #tempGblInfoDone1,
	                              error => #tempGblInfoError1,
	                              status => #tempGblInfoStatus1,
	                              DataRecord := #statDataRecord1);
	
	#statLPNDR_ReadGlobalInfo_DB2(execute := #statExecuteClock,
	                              hwId := #laddrProfinetPLC2,
	                              mode := 2,
	                              busy => #tempGblInfoBusy2,
	                              done => #tempGblInfoDone2,
	                              error => #tempGblInfoError2,
	                              status => #tempGblInfoStatus2,
	                              DataRecord := #statDataRecord2);
	
	IF #tempGblInfoError1 = TRUE THEN
	    #statError1 := TRUE;
	ELSE
	    #statError1 := FALSE;
	END_IF;
	
	#IEC_Timer_0_Instance_2(IN:=#statError1,
	                        PT:=T#10ms,
	                        Q=>#statChoose1);
	
	IF #tempGblInfoError2 = TRUE THEN
	    #statError2 := TRUE;
	ELSE
	    #statError2 := FALSE;
	END_IF;
	
	#IEC_Timer_0_Instance_3(IN := #statError2,
	                        PT := T#10ms,
	                        Q => #statChoose2);
	
	
	
	IF #statDataRecord1.mrpRole = 3 AND #statChoose1 = FALSE THEN
	    // Statement section IF
	    #statLPNDR_ReadMrpState := #laddrProfinetPLC1;
	    #statUndefinedState := FALSE;
	ELSIF #statDataRecord2.mrpRole = 3 AND #statChoose2 = FALSE THEN
	    #statLPNDR_ReadMrpState := #laddrProfinetPLC2;
	    #statUndefinedState := FALSE;
	ELSE
	    #statUndefinedState := TRUE;
	    
	END_IF;
	
	
	IF #statExecuteClock = FALSE THEN
	    #statToggleExecuteClock := TRUE;
	ELSE
	    ;
	END_IF;
	
	#IEC_Timer_0_Instance(IN := #statToggleExecuteClock,
	                      PT := T#5ms,
	                      Q => #statExecuteClock);
	
	IF #statExecuteClock = TRUE THEN
	    #statToggleExecuteClock := FALSE;
	ELSE
	    ;
	END_IF;
	
	IF #statExecuteClock2 = False AND #statUndefinedState = FALSE THEN
	    #statToggleExecuteClock2 := TRUE;
	ELSE
	    ;
	END_IF;
	
	#IEC_Timer_0_Instance_1(IN:=#statToggleExecuteClock2,
	                        PT:=T#5ms,
	                        Q=>#statExecuteClock2);
	
	IF #statExecuteClock2 = TRUE THEN
	    #statToggleExecuteClock2 := FALSE;
	ELSE
	    ;
	END_IF;
	
	#statLPNDR_ReadMrpState_DB(execute := #statExecuteClock2,
	                           hwId := #statLPNDR_ReadMrpState,
	                           busy => #tempMrpBusy,
	                           done => #tempMrpDone,
	                           error => #tempMrpError,
	                           mrpRingState => #mrpRingState,
	                           status => #tempMrpStatus);
	
	IF #statUndefinedState = TRUE THEN
	    #mrpRingState := 2;
	ELSE
	    ;
	END_IF;
	
END_FUNCTION_BLOCK

FUNCTION_BLOCK "plcStateEvaluation"
{ S7_Optimized_Access := 'TRUE' }
VERSION : 0.1
   VAR_INPUT 
      primaryID : Int;
      plc1OperationState : UInt;
      plc2OperationState : UInt;
      plcOperationStateSystem : UInt;
      plcMrpRingState : UInt;
   END_VAR

   VAR_OUTPUT 
      PLC_OperateStatus : Int;
      PLC_MrpState : Int;
      PLC1_LEDStatus : Int;
      PLC2_LEDStatus : Int;
   END_VAR

   VAR_IN_OUT 
      PLC12_StopMonitoring : Int;
   END_VAR

   VAR 
      statPrimaryID : Int;
      statPlc1State : UInt;
      statPlc2State : UInt;
      statPlcStateSystem : UInt;
      statPlcMrpRingState : UInt;
      statPlcStatus : Int;
      statPLC12StopMonitoring : Int;
   END_VAR


BEGIN
	//Wertzuweisung
	//
	
	#statPrimaryID := #primaryID;
	#statPlc1State := #plc1OperationState;
	#statPlc2State := #plc2OperationState;
	#statPlcStateSystem:= #plcOperationStateSystem;
	#statPlcMrpRingState := #plcMrpRingState;
	#PLC12_StopMonitoring := #statPLC12StopMonitoring;
	
	//PLC1 Status 
	// 
	CASE #statPlc1State OF 
	    1:  #PLC1_LEDStatus:= 1 //Synchronisiert
	        ;
	    4:
	        #PLC1_LEDStatus := 2 //Stop
	        ;
	    8:
	        #PLC1_LEDStatus := 3   //RUN-Solo
	        ;
	    9:
	        #PLC1_LEDStatus := 4   //RUN-Redundant
	        ;
	    21:
	        #PLC1_LEDStatus := 5   //Run-Syncup
	        ;
	    22:
	        #PLC1_LEDStatus := 6   //SYNCUP (nur die Backup PLC in SYNCUP)
	        ;
	    31:
	        #PLC1_LEDStatus := 7   //Zustand der Partner PLC unbekannt (z. B. wenn nicht erreichbar)
	        ;
	    37:
	        #PLC1_LEDStatus := 8   //RUN-Solo
	        ;
	    40:
	        #PLC1_LEDStatus := 9   //RUN-Redundant
	        ;
	    ELSE
	        #PLC1_LEDStatus := 10   //Details siehe Doku
	        ;
	END_CASE;
	
	
	//PLC2 Status 
	// 
	CASE #statPlc2State OF
	    1:
	        #PLC2_LEDStatus := 1 //Synchronisiert
	        ;
	    4:
	        #PLC2_LEDStatus := 2 //Stop
	        ;
	    8:
	        #PLC2_LEDStatus := 3   //RUN-Solo
	        ;
	    9:
	        #PLC2_LEDStatus := 4   //RUN-Redundant
	        ;
	    21:
	        #PLC2_LEDStatus := 5   //Run-Syncup
	        ;
	    22:
	        #PLC2_LEDStatus := 6   //SYNCUP (nur die Backup PLC in SYNCUP)
	        ;
	    31:
	        #PLC2_LEDStatus := 7   //Zustand der Partner PLC unbekannt (z. B. wenn nicht erreichbar)
	        ;
	    37:
	        #PLC2_LEDStatus := 8   //RUN-Solo
	        ;
	    40:
	        #PLC2_LEDStatus := 9   //RUN-Redundant
	        ;
	    ELSE
	        #PLC1_LEDStatus := 10   //Details siehe Doku
	        ;
	END_CASE;
	
	
	//PLC 1/2 Betriebszustand
	//
	IF #statPrimaryID = 1 THEN
	    #PLC_OperateStatus := 1;    //PLC1 Primary
	END_IF;
	
	IF #statPrimaryID = 2 THEN
	    #PLC_OperateStatus := 2;    //PLC2 Primary
	END_IF;
	
	
	//MRP-Ring
	//
	CASE #statPlcMrpRingState OF
	    0:
	        #PLC_MrpState := 0 //Ring Offen
	        ;
	    1:
	        #PLC_MrpState := 1 //Ring geschlossen
	        ;
	    2:
	        #PLC_MrpState := 2   //Zustand undefiniert
	        ;
	END_CASE;
	
	
	//Auswertung beide CPUen in Stop
	//
	#statPLC12StopMonitoring := 200;    //Konstante, die durch ein Skript im HMI zurückgesetzt wird
END_FUNCTION_BLOCK

ORGANIZATION_BLOCK "Main_Switch"   // OB123, LAD, ProgramCycle
TITLE = "Main Program Sweep (Cycle)"
{ S7_Optimized_Access := 'TRUE' }
// stored: AutoNumber false, SetENOAutomatically false
   VAR_INPUT
      Initial_Call : Bool;   // Initial call of this OB
      Remanence : Bool;   // =True, if remanent data are available
   END_VAR
   VAR_TEMP
      retvalue : Int;
      text : String;
      retVal : Word;
      Busy : Bool;
   END_VAR
   VAR_TEMP   // added for the SCL form of the ladder/FBD networks
      _w1 : Bool;
   END_VAR
BEGIN

REGION Network 1: Cycle Measurement - Tic
   // Scan and store but only to reset the runtime counter at the top of the scan. the Ret_Val is collected at the end of the program cycle or area of focus.
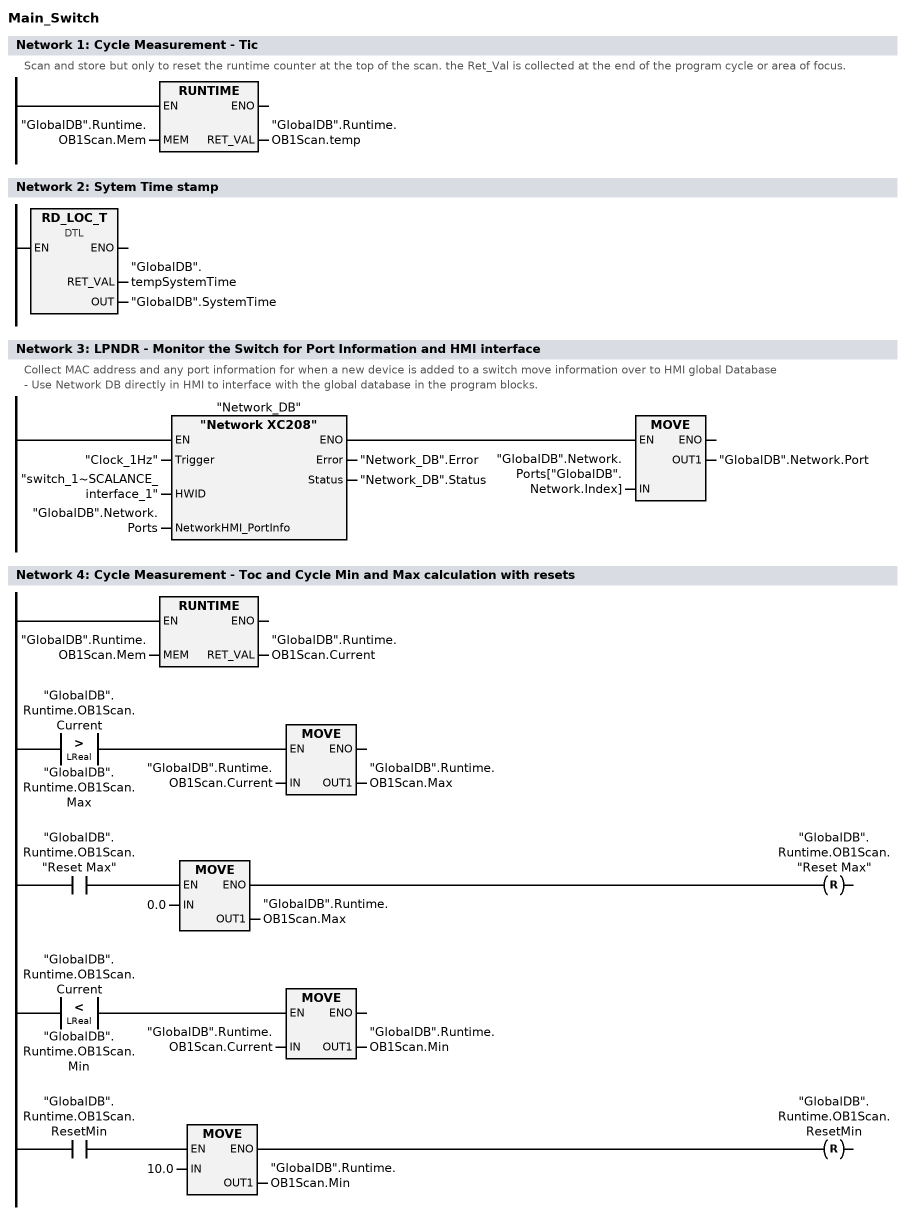
   // no SCL statement known for Runtime: written as a call
   "GlobalDB".Runtime.OB1Scan.temp := Runtime(mem := "GlobalDB".Runtime.OB1Scan.Mem);
END_REGION

REGION Network 2: Sytem Time stamp
   RUNG wire#powerrail
      { S7_Templates := "date_type := DTL" } RD_LOC_T(RET_VAL => "GlobalDB".tempSystemTime, OUT => "GlobalDB".SystemTime)
   END_RUNG
   // the same network as SCL:
   "GlobalDB".tempSystemTime := RD_LOC_T(OUT => "GlobalDB".SystemTime);
END_REGION

REGION Network 3: LPNDR - Monitor the Switch for Port Information and HMI interface
   // Collect MAC address and any port information for when a new device is added to a switch move information over to HMI global Database
   // 
   // - Use Network DB directly in HMI to interface with the global database in the program blocks.
   RUNG wire#powerrail
      "Network_DB"(Trigger := "Clock_1Hz", HWID := "switch_1~SCALANCE_interface_1", NetworkHMI_PortInfo := "GlobalDB".Network.Ports, Error => "Network_DB".Error, Status => "Network_DB".Status)
      Move(in := "GlobalDB".Network.Ports["GlobalDB".Network.Index], out1 => "GlobalDB".Network.Port)
   END_RUNG
   // the same network as SCL:
   "Network_DB"(Trigger := "Clock_1Hz",   // "Network XC208"
                HWID := "switch_1~SCALANCE_interface_1",
                NetworkHMI_PortInfo := "GlobalDB".Network.Ports,
                Error => "Network_DB".Error,
                Status => "Network_DB".Status,
                ENO => #_w1);
   IF #_w1 THEN "GlobalDB".Network.Port := "GlobalDB".Network.Ports["GlobalDB".Network.Index]; END_IF;
END_REGION

REGION Network 4: Cycle Measurement - Toc and Cycle Min and Max calculation with resets
   // no SCL statement known for Runtime: written as a call
   "GlobalDB".Runtime.OB1Scan.Current := Runtime(mem := "GlobalDB".Runtime.OB1Scan.Mem);
   IF "GlobalDB".Runtime.OB1Scan.Current > "GlobalDB".Runtime.OB1Scan.Max THEN
       "GlobalDB".Runtime.OB1Scan.Max := "GlobalDB".Runtime.OB1Scan.Current;
   END_IF;
   IF "GlobalDB".Runtime.OB1Scan."Reset Max" THEN
       "GlobalDB".Runtime.OB1Scan.Max := 0.0;
       "GlobalDB".Runtime.OB1Scan."Reset Max" := FALSE;
   END_IF;
   IF "GlobalDB".Runtime.OB1Scan.Current < "GlobalDB".Runtime.OB1Scan.Min THEN
       "GlobalDB".Runtime.OB1Scan.Min := "GlobalDB".Runtime.OB1Scan.Current;
   END_IF;
   IF "GlobalDB".Runtime.OB1Scan.ResetMin THEN
       "GlobalDB".Runtime.OB1Scan.Min := 10.0;
       "GlobalDB".Runtime.OB1Scan.ResetMin := FALSE;
   END_IF;
END_REGION
END_ORGANIZATION_BLOCK

FUNCTION_BLOCK "Network XC208"   // FB10, LAD
{ S7_Optimized_Access := 'TRUE' }
// stored: MemoryReserve 100, SetENOAutomatically false
   VAR_INPUT
      Trigger : Bool;   // Trigger the network scan for port info, rising edge
      HWID : HW_ANY;   // Scalance Interface of the switch
   END_VAR
   VAR_OUTPUT
      Error : Bool;
      Status : Word;
   END_VAR
   VAR_IN_OUT
      NetworkHMI_PortInfo : Variant;   // HMI input and output interface
   END_VAR
   VAR
      PortInformation { S7_SetPoint := 'True'} : "LPNDR_ReadGlobalInfo";   // LPNDR mode returns Port Information
   END_VAR
   VAR CONSTANT
      modeInterfaceInformation : Int := 1;
      modeMRPInformation : Int := 2;
      modePortInformation : Int := 3;
      modePortLinkStatus : Int := 4;
      modePortStatistics : Int := 5;
   END_VAR
BEGIN

REGION Network 1: Mode 3: Read Port Information
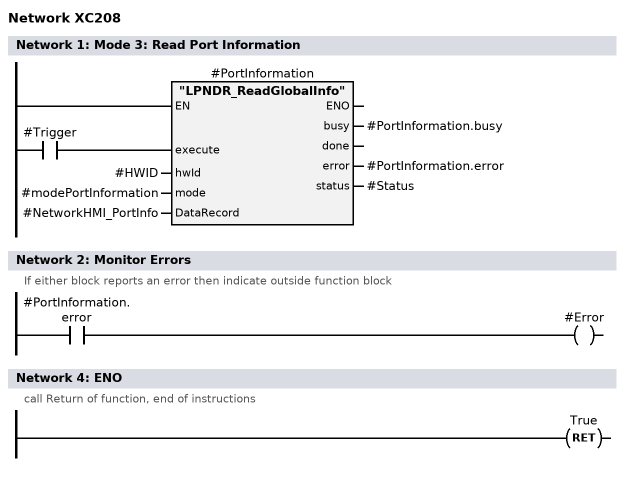
   RUNG wire#powerrail
      #PortInformation(execute := wire#w1, hwId := #HWID, mode := #modePortInformation, DataRecord := #NetworkHMI_PortInfo, busy => #PortInformation.busy, done =>, error => #PortInformation.error, status => #Status)
   END_RUNG
   RUNG wire#powerrail
      Contact( #Trigger )
   END_RUNG wire#w1
   // the same network as SCL:
   #PortInformation(execute := #Trigger,   // "LPNDR_ReadGlobalInfo"
                    hwId := #HWID,
                    mode := #modePortInformation,
                    DataRecord := #NetworkHMI_PortInfo,
                    busy => #PortInformation.busy,
                    error => #PortInformation.error,
                    status => #Status);
END_REGION

REGION Network 2: Monitor Errors
   // If either block reports an error then indicate outside function block
   RUNG wire#powerrail
      Contact( #PortInformation.error )
      Coil( #Error )
   END_RUNG
   // the same network as SCL:
   #Error := #PortInformation.error;
END_REGION

REGION Network 3
   // #Port."Port" := #Port.Ports[#Index];
END_REGION

REGION Network 4: ENO
   // call Return of function, end of instructions
   ENO := True;
   RETURN;
END_REGION
END_FUNCTION_BLOCK

FUNCTION "Move MAC" : Void   // FC11, LAD
{ S7_Optimized_Access := 'TRUE' }
// stored: SetENOAutomatically false
   VAR_INPUT
      InMAC : Array[0..5] of Byte;
   END_VAR
   VAR_OUTPUT
      OutMAC : Array[0..5] of Byte;
   END_VAR
BEGIN

REGION Network 1
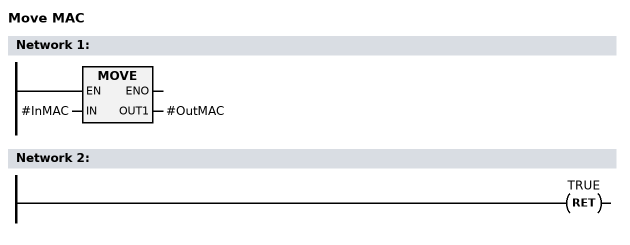
   RUNG wire#powerrail
      Move(in := #InMAC, out1 => #OutMAC)
   END_RUNG
   // the same network as SCL:
   #OutMAC := #InMAC;
END_REGION

REGION Network 2
   RUNG wire#powerrail
      ReturnCoil( TRUE )
   END_RUNG
   // the same network as SCL:
   ENO := TRUE;
   RETURN;
END_REGION
END_FUNCTION

FUNCTION_BLOCK "NetworkSwitchFaceplate"   // FB11, LAD
{ S7_Optimized_Access := 'TRUE' }
// stored: MemoryReserve 100, SetENOAutomatically false
   VAR_INPUT
      Index : Int;
   END_VAR
   VAR_OUTPUT
      PeerName { ExternalAccessible := 'False'; ExternalVisible := 'False'; ExternalWritable := 'False'} : String;
   END_VAR
   VAR_IN_OUT
      Port : "NetworkSwitchHMI";
   END_VAR
BEGIN

REGION Network 1 (SCL): Move all IN/OUT variables into Static values based on index selected from HMI

   #Port.Port := #Port.Ports[#Index];
END_REGION
END_FUNCTION_BLOCK

FUNCTION "EnS_Adv_CycInt200msFC" : Void
TITLE = FC for advanced data in cyclic interrupt OB
{ S7_Optimized_Access := 'TRUE' }
AUTHOR : Siemens
FAMILY : EnS
VERSION : 1.0
//FC for advanced data in cyclic interrupt OB

BEGIN
	
	//Advanced data collection 
	"InfeedPAC3200_Adv"(energyMeta := "InfeedPAC3200".energyMeta,
	                    orgData := "EnS_Org_CycInt200ms".orgData,
	                    advData := "pac3200_Adv_InfeedPAC3200".advData);
	
	//Advanced min/max data collection
	"InfeedPAC3200_AdvMinMax"(advDataMin := "pac3200_AdvMinMax_InfeedPAC3200".advDataMin,
	                          advDataMax := "pac3200_AdvMinMax_InfeedPAC3200".advDataMax);
	
END_FUNCTION

FUNCTION "EnS_Archive_CycInt500msFC" : Void
TITLE = FC for archiving functionality in cyclic interrupt OB
{ S7_Optimized_Access := 'TRUE' }
AUTHOR : Siemens
FAMILY : EnS
VERSION : 1.0
//FC for archiving functionality in cyclic interrupt OB

BEGIN
	
	//Archiving of buffer to HMI
	"EnS_Archive32469"(sD := "EnS_Archive32469".status,
	                   orgData := "EnS_Org_CycInt500ms".orgData,
	                   bufferWork := "EnS_BufferWork32469");
	
END_FUNCTION

FUNCTION "EnS_Basic_CycInt1sFC" : Void
TITLE = FC for basic data of measuring points in cyclic interrupt OB
{ S7_Optimized_Access := 'TRUE' }
AUTHOR : Siemens
FAMILY : EnS
VERSION : 1.0
//FC for basic data of measuring points in cyclic interrupt OB

BEGIN
	
	//Basic energy data
	//Calculation and data collection of periodic accumulated energy and average power
	"EnS_Calc_InfeedPAC3200"(power := "pac3200_InfeedPAC3200".power,
	                         energy := "pac3200_InfeedPAC3200".energy,
	                         orgData := "EnS_Org_CycInt1s".orgData,
	                         syncData := "EnS_Sync_Period_1".syncData,
	                         energyMeta := "InfeedPAC3200".energyMeta);
	
	//Basic data collection
	"InfeedPAC3200"(energyBasic := "EnS_Calc_InfeedPAC3200".energyBasic,
	                bufferDB := "EnS_Buffer32469",
	                sD := "InfeedPAC3200".energyMeta.id,
	                orgData := "EnS_Org_CycInt1s".orgData,
	                bufferWork := "EnS_BufferWork32469");
	
END_FUNCTION

ORGANIZATION_BLOCK "EnS_CycInt1sOB"
TITLE = Cyclic interrupt OB of 1s
{ S7_Optimized_Access := 'TRUE' }
AUTHOR : Siemens
FAMILY : EnS
VERSION : 1.0
//Cyclic interrupt OB of 1s

BEGIN
	//FC for organizational data in cyclic interrupt OB
	"EnS_Org_CycInt1sFC"();
	//FC for driver functionality of measuring points in cyclic interrupt OB
	"EnS_Drv_CycInt1sFC"();
	//FC for basic data of measuring points in cyclic interrupt OB
	"EnS_Basic_CycInt1sFC"();
	
END_ORGANIZATION_BLOCK

FUNCTION "EnS_Org_CycInt1sFC" : Void
TITLE = FC for organizational data in cyclic interrupt OB
{ S7_Optimized_Access := 'TRUE' }
AUTHOR : Siemens
FAMILY : EnS
VERSION : 1.0
//FC for organizational data in cyclic interrupt OB

BEGIN
	
	//Organizational data for cyclic interrupt OB
	"EnS_Org_CycInt1s"();
	
END_FUNCTION

FUNCTION "EnS_Drv_CycInt1sFC" : Void
TITLE = FC for driver functionality of measuring points in cyclic interrupt OB
{ S7_Optimized_Access := 'TRUE' }
AUTHOR : Siemens
FAMILY : EnS
VERSION : 1.0
//FC for driver functionality of measuring points in cyclic interrupt OB

BEGIN
	
	//Driver Functionality for basic value
	"pac3200_InfeedPAC3200"(orgData := "EnS_Org_CycInt1s".orgData,
	                        energyMeta := "InfeedPAC3200".energyMeta);
	
END_FUNCTION

ORGANIZATION_BLOCK "EnS_CycInt200msOB"
TITLE = Cyclic interrupt OB of 200ms
{ S7_Optimized_Access := 'TRUE' }
AUTHOR : Siemens
FAMILY : EnS
VERSION : 1.0
//Cyclic interrupt OB of 200ms

BEGIN
	//FC for organizational data in cyclic interrupt OB
	"EnS_Org_CycInt200msFC"();
	//FC for driver advanced functionality of measuring points in cyclic interrupt OB
	"EnS_DrvAdv_CycInt200msFC"();
	//FC for advanced data in cyclic interrupt OB
	"EnS_Adv_CycInt200msFC"();
	
END_ORGANIZATION_BLOCK

FUNCTION "EnS_Org_CycInt200msFC" : Void
TITLE = FC for organizational data in cyclic interrupt OB
{ S7_Optimized_Access := 'TRUE' }
AUTHOR : Siemens
FAMILY : EnS
VERSION : 1.0
//FC for organizational data in cyclic interrupt OB

BEGIN
	
	//Organizational data for cyclic interrupt OB
	"EnS_Org_CycInt200ms"();
	
END_FUNCTION

FUNCTION "EnS_DrvAdv_CycInt200msFC" : Void
TITLE = FC for driver advanced functionality of measuring points in cyclic interrupt OB
{ S7_Optimized_Access := 'TRUE' }
AUTHOR : Siemens
FAMILY : EnS
VERSION : 1.0
//FC for driver advanced functionality of measuring points in cyclic interrupt OB

BEGIN
	
	//Driver functionality for advanced energy data
	"pac3200_Adv_InfeedPAC3200"(orgData := "EnS_Org_CycInt200ms".orgData,
	                            energyMeta := "InfeedPAC3200".energyMeta,
	                            requestBufferHeader := "LAcycCom_RequestBuffer"."header",
	                            requestBufferElements := "LAcycCom_RequestBuffer"."elements",
	                            enableDrvAdv := "pac3200_InfeedPAC3200".enableDrvAdv,
	                            measData := "pac3200_InfeedPAC3200".measData);
	
	//Driver Functionality for advanced energy data with min/max value
	"pac3200_AdvMinMax_InfeedPAC3200"(orgData := "EnS_Org_CycInt200ms".orgData,
	                                  energyMeta := "InfeedPAC3200".energyMeta,
	                                  requestBufferHeader := "LAcycCom_RequestBuffer"."header",
	                                  requestBufferElements := "LAcycCom_RequestBuffer"."elements",
	                                  enableDrvAdv := "pac3200_InfeedPAC3200".enableDrvAdv,
	                                  measData := "pac3200_InfeedPAC3200".measData);
	
END_FUNCTION

ORGANIZATION_BLOCK "EnS_CycInt500msOB"
TITLE = Cyclic interrupt OB of 500ms
{ S7_Optimized_Access := 'TRUE' }
AUTHOR : Siemens
FAMILY : EnS
VERSION : 1.0
//Cyclic interrupt OB of 500ms

BEGIN
	//FC for organizational data in cyclic interrupt OB
	"EnS_Org_CycInt500msFC"();
	//FC for time synchronization in cyclic interrupt OB
	"EnS_Sync_CycInt500msFC"();
	//FC for archiving functionality in cyclic interrupt OB
	"EnS_Archive_CycInt500msFC"();
	
END_ORGANIZATION_BLOCK

FUNCTION "EnS_Org_CycInt500msFC" : Void
TITLE = FC for organizational data in cyclic interrupt OB
{ S7_Optimized_Access := 'TRUE' }
AUTHOR : Siemens
FAMILY : EnS
VERSION : 1.0
//FC for organizational data in cyclic interrupt OB

BEGIN
	
	//Organizational data for cyclic interrupt OB
	"EnS_Org_CycInt500ms"();
	
END_FUNCTION

FUNCTION "EnS_Sync_CycInt500msFC" : Void
TITLE = FC for time synchronization in cyclic interrupt OB
{ S7_Optimized_Access := 'TRUE' }
AUTHOR : Siemens
FAMILY : EnS
VERSION : 1.0
//FC for time synchronization in cyclic interrupt OB

BEGIN
	
	//Time synchroniztion for period
	"EnS_Sync_Period_1"(orgData := "EnS_Org_CycInt500ms".orgData);
	
END_FUNCTION

ORGANIZATION_BLOCK "EnS_LAcycCom_MainOB"
TITLE = Acyclic Communication OB
{ S7_Optimized_Access := 'TRUE' }
AUTHOR : Siemens
FAMILY : EnS
VERSION : 1.0
//Acyclic Communication OB

BEGIN
	//FC for LAcycCom ResourceManager Variant
	"EnS_LAcycCom_ResourceManagerFC"();
	
END_ORGANIZATION_BLOCK

FUNCTION "EnS_LAcycCom_ResourceManagerFC" : Void
TITLE = FC for LAcycCom ResourceManager Variant
{ S7_Optimized_Access := 'TRUE' }
AUTHOR : Siemens
FAMILY : EnS
VERSION : 1.0
//FC for LAcycCom ResourceManager Variant

BEGIN
	
	//LAcycCom ResourceManager Variant
	"EnS_LAcycCom_ResourceManager"(enable := True,
	                               requestBufferHeader := "LAcycCom_RequestBuffer"."header",
	                               requestBufferElements := "LAcycCom_RequestBuffer"."elements");
	
END_FUNCTION

FUNCTION "EnS_StartupFC" : Void
TITLE = FC for startup OB
{ S7_Optimized_Access := 'TRUE' }
AUTHOR : Siemens
FAMILY : EnS
VERSION : 1.0
//FC for startup OB

BEGIN
	
	//Organizational data for cyclic interrupt OB
	"EnS_Org_CycInt500ms"();
	
	//Organizational data for cyclic interrupt OB
	"EnS_Org_CycInt1s"();
	
	//Organizational data for cyclic interrupt OB
	"EnS_Org_CycInt200ms"();
	
END_FUNCTION

ORGANIZATION_BLOCK "EnS_StartupOB"
TITLE = Startup OB
{ S7_Optimized_Access := 'TRUE' }
AUTHOR : Siemens
FAMILY : EnS
VERSION : 1.0
//Startup OB

BEGIN
	//FC for startup OB
	"EnS_StartupFC"();
	
END_ORGANIZATION_BLOCK

FUNCTION_BLOCK "LPNDR_ReadGlobalInfo_2"
{ S7_Optimized_Access := 'TRUE' }
VERSION : 0.1
   VAR_INPUT 
      execute : Bool;
      hwId : HW_IO;
      mode : Int;
   END_VAR

   VAR_OUTPUT 
      busy : Bool;
      done : Bool;
      error : Bool;
      status : Word;
   END_VAR

   VAR_IN_OUT 
      DataRecord : Variant;
   END_VAR

   VAR 
      InstReadRecord {InstructionName := 'RDREC'; LibVersion := '1.0'} : RDREC;
      statReadRecord { ExternalAccessible := 'False'; ExternalVisible := 'False'; ExternalWritable := 'False'} : Array[0..4175] of Byte;
      statReadRecordLength : UInt;
      statReadRecordRequest : Bool;
      statOldExecute : Bool;
      statPDInterfaceMrpDataReal : UInt;
      statPDPortMrpDataReal : UInt;
      statPDInterfaceDataReal : UInt;
      statPDPortDataReal : UInt;
      statPDPortStatistic : UInt;
      statUnknown : UInt;
      statInterfaceInformation : "LPNDR_typeInterfaceInformation";
      statPortInformation : Array[1..52] of "LPNDR_typePortInformation";
      statPortLinkState : Array[1..52] of "LPNDR_typePortLinkState";
      statPortStatistic : Array[1..52] of "LPNDR_typePortStatistic";
      statBusy { S7_SetPoint := 'True'} : Bool;
   END_VAR

   VAR_TEMP 
      i : DInt;
      tempDataWord : Word;
      tempDataDWord : DWord;
      tempIndex : DInt;
      tempReturnValue : Int;
      tempPortNumber : USInt;
      tempNextMultipleBlockIndex : DInt;
      tempNextSubBlockIndex : DInt;
      tempState : Int;
      tempStatus : Word;
   END_VAR

   VAR CONSTANT 
      INVALID_TYPE_DATA_RECORD : Word := 16#5000;
      INVALID_MODE : Word := 16#5001;
      INVALID_ARRAY_TOO_SMALL : Word := 16#5002;
   END_VAR


BEGIN
	IF #execute <> #statOldExecute THEN
	  #statOldExecute := #execute;
	  
	  IF #statOldExecute THEN //positive edge
	    #statReadRecordRequest := true;
	    
	    #statReadRecordLength := 0;
	    
	    #status := 0;
	    #statBusy := true;
	    #done := false;
	    #error := false;
	  END_IF;
	END_IF;
	IF NOT #execute
	    AND NOT #statBusy
	THEN
	    #status := 0;
	    #statBusy := 0;
	    #done := false;
	    #error := false;
	END_IF;
	
	#InstReadRecord(REQ := #statReadRecordRequest,
	                ID := #hwId,
	                INDEX := 16#F841, //PDDataReal
	                MLEN := 0,
	                RECORD := #statReadRecord);
	
	IF #InstReadRecord.VALID THEN
	  #statReadRecordLength := #InstReadRecord.LEN;
	  
	  //init
	 #statPDPortDataReal := 0;
	#statPDInterfaceMrpDataReal := 0;
	#statPDPortMrpDataReal := 0;
	#statPDInterfaceDataReal := 0;
	 #statPDPortStatistic := 0;
	#statUnknown := 0;
	  //get data
	  //#tempIndex := 0; //get 1st BlockType
	  #tempPortNumber := 0;
	  WHILE (#tempIndex < #statReadRecordLength) DO
	    #tempReturnValue := READ_BIG(src_array := #statReadRecord,
	                                 dest_Variable => #tempDataWord,
	                                 pos := #tempIndex);
	    IF #tempDataWord = 16#0400 THEN //BlockType = MultipleBlockHeader
	      //get multiple block length
	      #tempReturnValue := READ_BIG(src_array := #statReadRecord,
	                                   dest_Variable => #tempDataWord,
	                                   pos := #tempIndex);
	      #tempNextMultipleBlockIndex := #tempIndex + #tempDataWord; //BlockLength + 4 bytes (BlockType + BlockLength); #tempIndex = 4
	      
	      //next BlockType
	      #tempIndex := #tempIndex + 12;
	      WHILE (#tempIndex < #tempNextMultipleBlockIndex) DO
	        //get sub block length
	        #tempIndex := #tempIndex + 2;
	        #tempReturnValue := READ_BIG(src_array := #statReadRecord,
	                                     dest_Variable => #tempDataWord,
	                                     pos := #tempIndex);
	        #tempNextSubBlockIndex := #tempIndex + #tempDataWord; //BlockLength + 4 bytes (BlockType + BlockLength); #tempIndex = 4
	        
	        //block type
	        #tempIndex := #tempIndex - 4;
	        #tempReturnValue := READ_BIG(src_array := #statReadRecord,
	                                     dest_Variable => #tempDataWord,
	                                     pos := #tempIndex);
	        CASE WORD_TO_INT(#tempDataWord) OF
	          16#020F: //PDPortDataReal
	            REGION PDPortDataReal
	            #statPDPortDataReal := #statPDPortDataReal + 1;
	              
	              //increase port number (index)
	              #tempPortNumber := #tempPortNumber + 1;
	              
	              //get own port ID
	              #tempIndex := #tempIndex + 10;
	              #tempDataWord := #statReadRecord[#tempIndex]; //number of characters
	              #tempIndex := #tempIndex + 1;
	              Chars_TO_Strg(Chars := #statReadRecord,
	                            pChars := #tempIndex,
	                            Cnt := MIN(IN1 := INT_TO_WORD(MAX_LEN(#statPortInformation[#tempPortNumber].portDiagnostic.portName)), IN2 := #tempDataWord),
	                            Strg => #statPortInformation[#tempPortNumber].portDiagnostic.portName);
	              #statPortLinkState[#tempPortNumber].portName := #statPortInformation[#tempPortNumber].portDiagnostic.portName;
	              //check if LLDP data is available
	              #tempIndex := #tempIndex + #tempDataWord;
	              IF #statReadRecord[#tempIndex] > 0 THEN
	                //adjust padding bytes
	                #tempDataDWord := (#tempDataWord + 6) MOD 4;
	                IF #tempDataDWord > 0 THEN
	                  #tempIndex := #tempIndex + (4 - DWORD_TO_WORD(#tempDataDWord));
	                END_IF;
	                
	                //get ID of remote port
	                #tempIndex := #tempIndex + 1;
	                #tempDataWord := #statReadRecord[#tempIndex]; //number of characters
	                #tempIndex := #tempIndex + 1;
	                Chars_TO_Strg(Chars := #statReadRecord,
	                              pChars := #tempIndex,
	                              Cnt := MIN(IN1 := INT_TO_WORD(MAX_LEN(#statPortInformation[#tempPortNumber].peerPortName)), IN2 := #tempDataWord),
	                              Strg => #statPortInformation[#tempPortNumber].peerPortName);
	                
	                //get name of remote station
	                #tempIndex := #tempIndex + #tempDataWord;
	                #tempDataWord := #statReadRecord[#tempIndex]; //number of characters
	                #tempIndex := #tempIndex + 1;
	                Chars_TO_Strg(Chars := #statReadRecord,
	                              pChars := #tempIndex,
	                              Cnt := #tempDataWord,
	                              Strg => #statPortInformation[#tempPortNumber].peerNameofStation);
	                
	                //get cable delay in nsec
	                #tempIndex := #tempIndex + #tempDataWord;
	                
	                //adjust padding bytes
	                #tempDataDWord := (#tempDataWord + 10) MOD 4;
	                IF #tempDataDWord > 0 THEN
	                  #tempIndex := #tempIndex + (4 - DWORD_TO_WORD(#tempDataDWord));
	                END_IF;
	                
	                #tempReturnValue := READ_BIG(src_array := #statReadRecord,
	                                             dest_Variable => #tempDataDWord,
	                                             pos := #tempIndex);
	                IF #tempDataDWord <> 0 THEN
	                    #statPortInformation[#tempPortNumber].lineDelay := DWORD_TO_UDINT(#tempDataDWord - 16#8000_0000);
	                ELSE
	                    #statPortInformation[#tempPortNumber].lineDelay:= 0;
	                END_IF;
	                
	                //get remote MAC address
	                FOR #i := 0 TO 5 BY 1 DO
	                    #statPortInformation[#tempPortNumber].peerMacAdress[5-#i] := #statReadRecord[#tempIndex + #i];
	                END_FOR;
	              ELSE
	                  #statPortInformation[#tempPortNumber].peerPortName:= '';
	                  #statPortInformation[#tempPortNumber].peerNameofStation:= '';
	                  #statPortInformation[#tempPortNumber].lineDelay:= 0;
	                FOR #i := 0 TO 5 BY 1 DO
	                    #statPortInformation[#tempPortNumber].peerMacAdress[#i] := 0;
	                END_FOR;
	              END_IF;
	              
	              //get MediaType
	              #tempIndex := #tempNextSubBlockIndex - 4; //count index backwards
	              #tempReturnValue := READ_BIG(src_array := #statReadRecord,
	                                           dest_Variable => #tempDataDWord,
	                                           pos := #tempIndex);
	              #statPortInformation[#tempPortNumber].mediaType := DWORD_TO_USINT(#tempDataDWord);
	              
	              //get PortState
	              #tempIndex := #tempIndex - 8;
	              #tempReturnValue := READ_BIG(src_array := #statReadRecord,
	                                           dest_Variable => #tempDataWord,
	                                           pos := #tempIndex);
	             
	              #statPortInformation[#tempPortNumber].portDiagnostic.portLinkState := #tempDataWord.%B0;
	              #statPortInformation[#tempPortNumber].portDiagnostic.portPortState := #tempDataWord.%B1;
	              #statPortLinkState[#tempPortNumber].portLinkState := #tempDataWord.%B0;
	              #statPortLinkState[#tempPortNumber].portPortState := #tempDataWord.%B1;
	                
	                //get MAUType
	                #tempIndex := #tempIndex - 14;
	                #tempReturnValue := READ_BIG(src_array := #statReadRecord,
	                                             dest_Variable => #tempDataWord,
	                                             pos := #tempIndex);
	                CASE WORD_TO_INT(#tempDataWord) OF
	                  16#0005, 16#000A, 16#000B, 16#000C, 16#000D:
	                      #statPortInformation[#tempPortNumber].dataRate := '10M';
	                  16#000F, 16#0010,  16#0011,  16#0012:
	                      #statPortInformation[#tempPortNumber].dataRate  := '100M';
	                  16#0015, 16#0016, 16#0018, 16#0019, 16#001A, 16#001D, 16#001E:
	                          #statPortInformation[#tempPortNumber].dataRate := '1G';
	                  16#002A:
	                      #statPortInformation[#tempPortNumber].dataRate  := '2M';
	                  16#002B:
	                      #statPortInformation[#tempPortNumber].dataRate := '10M';
	                  ELSE
	                    IF #tempDataWord > 16#004E THEN
	                        #statPortInformation[#tempPortNumber].dataRate := '0';
	                  
	                    ELSIF #tempDataWord >= 16#004B THEN
	                   #statPortInformation[#tempPortNumber].dataRate  := '100G';
	                    ELSIF #tempDataWord >= 16#0046 THEN
	                        #statPortInformation[#tempPortNumber].dataRate := '40G';
	                    ELSIF #tempDataWord >= 16#0041 THEN
	                        #statPortInformation[#tempPortNumber].dataRate  := '10G';
	                    ELSIF #tempDataWord >= 16#003B THEN
	                        #statPortInformation[#tempPortNumber].dataRate := '10G1G';
	                    ELSIF #tempDataWord >= 16#0038 THEN
	                        #statPortInformation[#tempPortNumber].dataRate := '1G';
	                    ELSIF #tempDataWord >= 16#0036 THEN
	                        #statPortInformation[#tempPortNumber].dataRate := '10G'; //todo: or 100BasePXFD, see PN spec
	                    ELSIF #tempDataWord >= 16#002F THEN
	                        #statPortInformation[#tempPortNumber].dataRate  := '1G';
	                    ELSIF #tempDataWord >= 16#002C THEN
	                        #statPortInformation[#tempPortNumber].dataRate := '100M';
	                    ELSIF #tempDataWord >= 16#001F THEN
	                        #statPortInformation[#tempPortNumber].dataRate  := '10G';
	                    ELSE
	                        #statPortInformation[#tempPortNumber].dataRate := '0';
	                    
	                    END_IF;
	            END_CASE;
	            END_REGION
	            
	          16#0212: //PDInterfaceMrpDataReal
	            REGION PDInterfaceMrpDataReal
	             #statPDInterfaceMrpDataReal := #statPDInterfaceMrpDataReal + 1;
	              
	              #tempIndex := #tempIndex + 5;
	              IF #statReadRecord[#tempIndex] = 1 THEN //number of MRP instances
	                //get MRP role
	                #tempIndex := #tempIndex + 25;
	                #tempReturnValue := READ_BIG(src_array := #statReadRecord,
	                                             dest_Variable => #tempDataWord,
	                                             pos := #tempIndex);
	                #statInterfaceInformation.mrp.mrpRole := WORD_TO_UINT(#tempDataWord);
	                
	                //get MRP domain name
	              IF #tempDataWord > 0 THEN
	                  #tempIndex := #tempIndex + 2;
	                  #tempDataWord := #statReadRecord[#tempIndex]; //number of characters
	                  #tempIndex := #tempIndex + 1;
	                  Chars_TO_Strg(Chars := #statReadRecord,
	                                pChars := #tempIndex,
	                                Cnt := #tempDataWord,
	                                Strg => #statInterfaceInformation.mrp.domainName);
	                ELSE
	                   #statInterfaceInformation.mrp.domainName:= '';
	               END_IF;
	                
	                //todo
	                //padding bytes
	                //MRP parameters, but for now this information is not helpful
	              END_IF;
	            END_REGION
	            
	          16#0215: //PDPortMrpDataReal
	            REGION PDPortMrpDataReal
	             #statPDPortMrpDataReal :=#statPDPortMrpDataReal + 1;
	            END_REGION
	            
	          16#0240: //PDInterfaceDataReal
	            REGION PDInterfaceDataReal
	             #statPDInterfaceDataReal := #statPDInterfaceDataReal + 1;
	              
	              //get device name
	              #tempIndex := #tempIndex + 4;
	              #tempDataWord := #statReadRecord[#tempIndex]; //number of characters
	              #tempIndex := #tempIndex + 1;
	              Chars_TO_Strg(Chars := #statReadRecord,
	                            pChars := #tempIndex,
	                            Cnt := #tempDataWord,
	                            Strg => #statInterfaceInformation.nameOfStation);
	              
	              #tempIndex := #tempIndex + #tempDataWord;
	              //adjust padding bytes
	              #tempDataDWord := (#tempDataWord + 7) MOD 4;
	              IF #tempDataDWord > 0 THEN
	                #tempIndex := #tempIndex + (4 - DWORD_TO_WORD(#tempDataDWord));
	              END_IF;
	              
	              //get local MAC address
	              FOR #i := 0 TO 5 BY 1 DO
	                  #statInterfaceInformation.macAddress[5 - #i] := #statReadRecord[#tempIndex + #i];
	              END_FOR;
	              
	              //get local IP address
	              #tempIndex := #tempIndex + 8; //6 bytes of MAC + 2 padding bytes
	              FOR #i := 0 TO 3 BY 1 DO
	                  #statInterfaceInformation.ipAdress[3 - #i] := #statReadRecord[#tempIndex + #i];
	              END_FOR;
	                
	              //get local subnetmask
	              #tempIndex := #tempIndex + 4;
	              FOR #i := 0 TO 3 BY 1 DO
	                  #statInterfaceInformation.subnetMask[3 - #i] := #statReadRecord[#tempIndex + #i];
	              END_FOR;
	              
	              //get local gateway
	              #tempIndex := #tempIndex + 4;
	              FOR #i := 0 TO 3 BY 1 DO
	                  #statInterfaceInformation.gateway[3 - #i] := #statReadRecord[#tempIndex + #i];
	              END_FOR;
	            END_REGION
	            
	          16#0251: //PDPortStatistic
	            REGION PDPortStatistic
	               #statPDPortStatistic := #statPDPortStatistic + 1;
	                IF #statPDPortStatistic > 1
	                THEN
	                    #tempIndex := #tempIndex + 6; //count index backwards
	                    #tempReturnValue := READ_BIG(src_array := #statReadRecord,
	                                                 dest_Variable => #statPortStatistic[#tempPortNumber].inOctets,
	                                                 pos := #tempIndex);
	                 
	                    #tempReturnValue := READ_BIG(src_array := #statReadRecord,
	                                                 dest_Variable => #statPortStatistic[#tempPortNumber].outOctets,
	                                                 pos := #tempIndex);
	                 
	                    #tempReturnValue := READ_BIG(src_array := #statReadRecord,
	                                                 dest_Variable => #statPortStatistic[#tempPortNumber].inDiscards,
	                                                 pos := #tempIndex);
	                  
	                    #tempReturnValue := READ_BIG(src_array := #statReadRecord,
	                                                 dest_Variable => #statPortStatistic[#tempPortNumber].outDiscards,
	                                                 pos := #tempIndex);
	                
	                    #tempReturnValue := READ_BIG(src_array := #statReadRecord,
	                                                 dest_Variable => #statPortStatistic[#tempPortNumber].inErrors,
	                                                 pos := #tempIndex);
	                    
	                    #tempReturnValue := READ_BIG(src_array := #statReadRecord,
	                                                 dest_Variable => #statPortStatistic[#tempPortNumber].outErrors,
	                                                 pos := #tempIndex);
	                ELSE
	                    ;
	                END_IF;
	                    
	            END_REGION
	            
	          ELSE
	            REGION BlockUnknown
	              #statUnknown := #statUnknown + 1;
	              //RETURN; //for testing
	            END_REGION
	        END_CASE;
	        
	        #tempIndex := #tempNextSubBlockIndex;
	      END_WHILE;
	      
	      #tempIndex := #tempNextMultipleBlockIndex;
	    ELSE
	      //todo
	      ; //error: no multiple block or wrong next index calculation
	    END_IF;
	  END_WHILE;
	  CASE #mode OF
	      1:
	          IF (TypeOf(#DataRecord) = LPNDR_typeInterfaceInformation) THEN
	                  #tempState := MOVE_BLK_VARIANT(SRC := #statInterfaceInformation, COUNT := 1, SRC_INDEX := 0, DEST_INDEX := 0, DEST => #DataRecord);
	         
	          ELSE
	              #tempState := WORD_TO_INT(#INVALID_TYPE_DATA_RECORD);
	          END_IF;
	      2:
	          IF (TypeOf(#DataRecord) = LPNDR_typeMrpInformation) THEN
	              #tempState := MOVE_BLK_VARIANT(SRC := #statInterfaceInformation.mrp, COUNT := 1, SRC_INDEX := 0, DEST_INDEX := 0, DEST => #DataRecord);
	          ELSE
	              #tempState := WORD_TO_INT(#INVALID_TYPE_DATA_RECORD);
	          END_IF;
	      3:
	          IF (TypeOfElements(#DataRecord) = LPNDR_typePortInformation) THEN
	              IF (CountOfElements(#DataRecord) > (#statPDPortDataReal - 2))
	              THEN
	                  #tempState := MOVE_BLK_VARIANT(SRC := #statPortInformation, COUNT := #statPDPortDataReal, SRC_INDEX := 0, DEST_INDEX := 0, DEST => #DataRecord);
	              ELSE
	                  #tempState := WORD_TO_INT(#INVALID_ARRAY_TOO_SMALL);
	              END_IF;
	          ELSE
	              #tempState := WORD_TO_INT(#INVALID_TYPE_DATA_RECORD);
	          END_IF;
	  4:
	      IF (TypeOfElements(#DataRecord) = LPNDR_typePortLinkState) THEN
	          IF (CountOfElements(#DataRecord)> (#statPDPortDataReal-2))
	              THEN
	                  #tempState := MOVE_BLK_VARIANT(SRC := #statPortLinkState, COUNT := #statPDPortDataReal, SRC_INDEX := 0, DEST_INDEX := 0, DEST => #DataRecord);
	              ELSE
	                  #tempState := WORD_TO_INT(#INVALID_ARRAY_TOO_SMALL);
	              END_IF;
	      ELSE
	          #tempState := WORD_TO_INT(#INVALID_TYPE_DATA_RECORD);
	      END_IF;
	  5:
	      IF (TypeOfElements(#DataRecord) = LPNDR_typePortStatistic) THEN
	          IF (CountOfElements(#DataRecord)> (#statPDPortStatistic-3))
	              THEN
	          #tempState := MOVE_BLK_VARIANT(SRC := #statPortStatistic, COUNT :=(#statPDPortStatistic-1), SRC_INDEX := 0, DEST_INDEX := 0, DEST => #DataRecord);
	              ELSE
	                  #tempState := WORD_TO_INT(#INVALID_ARRAY_TOO_SMALL);
	              END_IF;
	      ELSE
	          #tempState := WORD_TO_INT(#INVALID_TYPE_DATA_RECORD);
	      END_IF;
	      
	  ELSE
	          #tempState := WORD_TO_INT(#INVALID_MODE);
	  END_CASE;
	  IF (#tempState > 0) THEN
	      #statBusy := false;
	      #error := true;
	      #status := INT_TO_WORD(#tempState);
	  ELSE
	      #statBusy := false;
	      #done := true;
	  END_IF;
	  
	  #statReadRecordRequest := false;
	ELSIF #InstReadRecord.ERROR THEN
	    #tempStatus.%B0 := #InstReadRecord.STATUS.%B1;
	    #tempStatus.%B1 := #InstReadRecord.STATUS.%B2;
	    #status := #tempStatus;
	  #statBusy := false;
	  #error := true;
	  
	  #statReadRecordRequest := false;
	END_IF;
	#busy := #statBusy;
END_FUNCTION_BLOCK

DATA_BLOCK "R_H_Sys_Status_DB"   // DB50
// stored: AutoNumber false, InstanceOfName R_H_Sys_Status, InstanceOfType FB
"R_H_Sys_Status"
BEGIN
END_DATA_BLOCK

DATA_BLOCK "LRedIO_RedAI_DB"   // DB1
AUTHOR : SiemensAG
FAMILY : LRedIO
VERSION : 1.0
// stored: InstanceOfName LRedIO_RedAI, InstanceOfType FB
"LRedIO_RedAI"
   // VAR_INPUT
   //    redInput1 : DInt;
   //    redInput2 : DInt;
   //    valueStateCh1 : Bool;
   //    valueStateCh2 : Bool;
   //    outputValue : USInt;
   //    hysterese : Int;
   //    discrepancy : Real;
   //    discrepancyTime : Time;
   //    endOfMeasuringRange : DInt;
   //    substitutionValue : DInt;
   //    useSubstitutionValue : USInt;
   //    ack : Bool;
   // END_VAR
   // VAR_OUTPUT
   //    warning : Bool;
   //    error : Bool;
   //    ackReq : Bool;
   //    status : Word;
   //    output : DInt;
   // END_VAR
   // VAR
   //    statRedInput1 { ExternalAccessible := 'False'; ExternalVisible := 'False'; ExternalWritable := 'False'} : DInt;
   //    statRedInput2 { ExternalAccessible := 'False'; ExternalVisible := 'False'; ExternalWritable := 'False'} : DInt;
   //    statValuestateCh1 { ExternalAccessible := 'False'; ExternalVisible := 'False'; ExternalWritable := 'False'} : Bool;
   //    statValuestateCh2 { ExternalAccessible := 'False'; ExternalVisible := 'False'; ExternalWritable := 'False'} : Bool;
   //    statDiscrepancy { ExternalAccessible := 'False'; ExternalVisible := 'False'; ExternalWritable := 'False'} : Real;
   //    statValuestateBad1 { ExternalAccessible := 'False'; ExternalVisible := 'False'; ExternalWritable := 'False'} : Bool;
   //    statValuestateBad2 { ExternalAccessible := 'False'; ExternalVisible := 'False'; ExternalWritable := 'False'} : Bool;
   //    statAck { ExternalAccessible := 'False'; ExternalVisible := 'False'; ExternalWritable := 'False'} : Bool;
   //    statAckNec { ExternalAccessible := 'False'; ExternalVisible := 'False'; ExternalWritable := 'False'} : Bool;
   //    statState { ExternalAccessible := 'False'; ExternalVisible := 'False'; ExternalWritable := 'False'} : Int;
   //    statDiscError { ExternalAccessible := 'False'; ExternalVisible := 'False'; ExternalWritable := 'False'} : Bool;
   //    statOutputValue { ExternalAccessible := 'False'; ExternalVisible := 'False'; ExternalWritable := 'False'} : USInt;
   //    statWrongOutputValue { ExternalAccessible := 'False'; ExternalVisible := 'False'; ExternalWritable := 'False'} : Bool;
   //    statWrongDisc { ExternalAccessible := 'False'; ExternalVisible := 'False'; ExternalWritable := 'False'} : Bool;
   //    statWrongHysterese { ExternalAccessible := 'False'; ExternalVisible := 'False'; ExternalWritable := 'False'} : Bool;
   //    statHysterese { ExternalAccessible := 'False'; ExternalVisible := 'False'; ExternalWritable := 'False'} : Int;
   //    statInputDifference { ExternalAccessible := 'False'; ExternalVisible := 'False'; ExternalWritable := 'False'} : DInt;
   //    statAbsInputDifference { ExternalAccessible := 'False'; ExternalVisible := 'False'; ExternalWritable := 'False'} : DInt;
   //    statDiscrepancyCalc { ExternalAccessible := 'False'; ExternalVisible := 'False'; ExternalWritable := 'False'} : DInt;
   //    statHystereseCalc { ExternalAccessible := 'False'; ExternalVisible := 'False'; ExternalWritable := 'False'} : DInt;
   //    statHysteresecheckOK { ExternalAccessible := 'False'; ExternalVisible := 'False'; ExternalWritable := 'False'} : Bool;
   //    statEndOfMeasuringRange { ExternalAccessible := 'False'; ExternalVisible := 'False'; ExternalWritable := 'False'} : DInt;
   //    statWrongEndOfMeasuringRange { ExternalAccessible := 'False'; ExternalVisible := 'False'; ExternalWritable := 'False'} : Bool;
   //    statSubValue { ExternalAccessible := 'False'; ExternalVisible := 'False'; ExternalWritable := 'False'} : DInt;
   //    statUseSubstitutionValue { ExternalAccessible := 'False'; ExternalVisible := 'False'; ExternalWritable := 'False'} : USInt;
   //    statWrongSubValue { ExternalAccessible := 'False'; ExternalVisible := 'False'; ExternalWritable := 'False'} : Bool;
   //    statAckEdge { ExternalAccessible := 'False'; ExternalVisible := 'False'; ExternalWritable := 'False'} : Bool;
   //    statWrongUseSubVal { ExternalAccessible := 'False'; ExternalVisible := 'False'; ExternalWritable := 'False'} : Bool;
   //    statDiscrepancyTime { ExternalAccessible := 'False'; ExternalVisible := 'False'; ExternalWritable := 'False'} : Time;
   //    statStartDiscTime { ExternalAccessible := 'False'; ExternalVisible := 'False'; ExternalWritable := 'False'} : Bool;
   //    statInstDiscrepancyTime { ExternalAccessible := 'False'; ExternalVisible := 'False'; ExternalWritable := 'False'; S7_SetPoint := 'True'} : TON_TIME;
   //    statStatus { ExternalAccessible := 'False'; ExternalVisible := 'False'; ExternalWritable := 'False'} : Word;
   //    statWrongDiscTime { ExternalAccessible := 'False'; ExternalVisible := 'False'; ExternalWritable := 'False'} : Bool;
   //    statOutput { ExternalAccessible := 'False'; ExternalVisible := 'False'; ExternalWritable := 'False'} : DInt;
   //    statParamError { ExternalAccessible := 'False'; ExternalVisible := 'False'; ExternalWritable := 'False'} : Bool;
   //    statOldRedInput1 { ExternalAccessible := 'False'; ExternalVisible := 'False'; ExternalWritable := 'False'} : DInt;
   //    statOldRedInput2 { ExternalAccessible := 'False'; ExternalVisible := 'False'; ExternalWritable := 'False'} : DInt;
   //    statNewRedInput1 { ExternalAccessible := 'False'; ExternalVisible := 'False'; ExternalWritable := 'False'} : DInt;
   //    statNewRedInput2 { ExternalAccessible := 'False'; ExternalVisible := 'False'; ExternalWritable := 'False'} : DInt;
   //    statLastValidOut { ExternalAccessible := 'False'; ExternalVisible := 'False'; ExternalWritable := 'False'} : DInt;
   //    statStoreRisingEdge : Bool;
   //    statDiscrepancyTimeTrue : Bool;
   // END_VAR
BEGIN
END_DATA_BLOCK

DATA_BLOCK "fbPnPnCouplerRightDiag_DB"   // DB12
// stored: InstanceOfName fbGetDiagPnPnCouplerDiag, InstanceOfType FB
"fbGetDiagPnPnCouplerDiag"
BEGIN
END_DATA_BLOCK

DATA_BLOCK "fbPnPnLeftCouplerDiag_DB"   // DB13
// stored: InstanceOfName fbGetDiagPnPnCouplerDiag, InstanceOfType FB
"fbGetDiagPnPnCouplerDiag"
BEGIN
END_DATA_BLOCK

DATA_BLOCK "Network_DB"   // DB31
// stored: InstanceOfName Network XC208, InstanceOfType FB
"Network XC208"
BEGIN
END_DATA_BLOCK

DATA_BLOCK "instanceR_H_Sys_Status_DB"   // DB28
// stored: InstanceOfName R_H_Sys_Status, InstanceOfType FB
"R_H_Sys_Status"
BEGIN
END_DATA_BLOCK

DATA_BLOCK "plcStateEvaluation_DB"   // DB27
// stored: InstanceOfName plcStateEvaluation, InstanceOfType FB
"plcStateEvaluation"
BEGIN
END_DATA_BLOCK

DATA_BLOCK "plcStateEvaluation_DB_1"   // DB29
// stored: InstanceOfName plcStateEvaluation, InstanceOfType FB
"plcStateEvaluation"
BEGIN
END_DATA_BLOCK

DATA_BLOCK "FBR1_PNPortStatus_DB"   // DB25
// stored: InstanceOfName PN Port Status, InstanceOfType FB
"PN Port Status"
BEGIN
END_DATA_BLOCK

DATA_BLOCK "FBR2_PNPortStatus_DB"   // DB26
// stored: InstanceOfName PN Port Status, InstanceOfType FB
"PN Port Status"
BEGIN
END_DATA_BLOCK

DATA_BLOCK "Switch1P8_PNPortStatus_DB"   // DB20
// stored: InstanceOfName PN Port Status, InstanceOfType FB
"PN Port Status"
BEGIN
END_DATA_BLOCK

DATA_BLOCK "Switch1_P7_PNPortStatus_DB"   // DB30
// stored: InstanceOfName PN Port Status, InstanceOfType FB
"PN Port Status"
BEGIN
END_DATA_BLOCK

DATA_BLOCK "InfeedPAC3200"   // DB19
TITLE = Instance DB of basic data collection
// Instance DB of basic data collection
// stored: InstanceOfName EnS_EnergyDataBasic, InstanceOfType FB
"EnS_EnergyDataBasic"
   // VAR_INPUT
   //    energyMeta : "EnS_typeEnergyMeta";
   //    energyBasic : "EnS_typeEnergyBasic";
   //    bufferDB { ExternalAccessible := 'False'; ExternalVisible := 'False'; ExternalWritable := 'False'} : DB_ANY;
   //    sD : Variant;
   //    messageSuppress { ExternalAccessible := 'False'; ExternalVisible := 'False'; ExternalWritable := 'False'} : Bool;
   // END_VAR
   // VAR_OUTPUT
   //    error { ExternalAccessible := 'False'; ExternalVisible := 'False'; ExternalWritable := 'False'} : Bool;
   //    errorAlarm1 { ExternalAccessible := 'False'; ExternalVisible := 'False'; ExternalWritable := 'False'} : Bool;
   //    errorAlarm2 { ExternalAccessible := 'False'; ExternalVisible := 'False'; ExternalWritable := 'False'} : Bool;
   //    errorAlarm3 { ExternalAccessible := 'False'; ExternalVisible := 'False'; ExternalWritable := 'False'} : Bool;
   //    alarmState1 { ExternalAccessible := 'False'; ExternalVisible := 'False'; ExternalWritable := 'False'} : Byte;
   //    alarmState2 { ExternalAccessible := 'False'; ExternalVisible := 'False'; ExternalWritable := 'False'} : Byte;
   //    alarmState3 { ExternalAccessible := 'False'; ExternalVisible := 'False'; ExternalWritable := 'False'} : Byte;
   //    status { ExternalAccessible := 'False'; ExternalVisible := 'False'; ExternalWritable := 'False'} : Word;
   //    status1 { ExternalAccessible := 'False'; ExternalVisible := 'False'; ExternalWritable := 'False'} : Word;
   //    status2 { ExternalAccessible := 'False'; ExternalVisible := 'False'; ExternalWritable := 'False'} : Word;
   //    status3 { ExternalAccessible := 'False'; ExternalVisible := 'False'; ExternalWritable := 'False'} : Word;
   //    statusAlarm1 { ExternalAccessible := 'False'; ExternalVisible := 'False'; ExternalWritable := 'False'} : Word;
   //    statusAlarm2 { ExternalAccessible := 'False'; ExternalVisible := 'False'; ExternalWritable := 'False'} : Word;
   //    statusAlarm3 { ExternalAccessible := 'False'; ExternalVisible := 'False'; ExternalWritable := 'False'} : Word;
   // END_VAR
   // VAR_IN_OUT
   //    orgData : "EnS_typeOrgData";
   //    bufferWork : "EnS_typeBufferWork";
   // END_VAR
   // VAR
   //    Program_Alarm1 { ExternalAccessible := 'False'; ExternalVisible := 'False'; ExternalWritable := 'False'; S7_SetPoint := 'True'} : Program_Alarm;
   //    Program_Alarm2 { ExternalAccessible := 'False'; ExternalVisible := 'False'; ExternalWritable := 'False'; S7_SetPoint := 'True'} : Program_Alarm;
   //    Program_Alarm3 { ExternalAccessible := 'False'; ExternalVisible := 'False'; ExternalWritable := 'False'; S7_SetPoint := 'True'} : Program_Alarm;
   //    ss_BufferWrite { ExternalAccessible := 'False'; ExternalVisible := 'False'; ExternalWritable := 'False'; S7_SetPoint := 'True'} : "EnS_BufferWrite";
   //    ss_DataEnergy { ExternalAccessible := 'False'; ExternalVisible := 'False'; ExternalWritable := 'False'; S7_SetPoint := 'True'} : "EnS_typeBufferWriteCtrl";
   //    ss_DataPower { ExternalAccessible := 'False'; ExternalVisible := 'False'; ExternalWritable := 'False'; S7_SetPoint := 'True'} : "EnS_typeBufferWriteCtrl";
   //    ss_DataEnergyCounter { ExternalAccessible := 'False'; ExternalVisible := 'False'; ExternalWritable := 'False'; S7_SetPoint := 'True'} : "EnS_typeBufferWriteCtrl";
   //    si16_CycleWrite { ExternalAccessible := 'False'; ExternalVisible := 'False'; ExternalWritable := 'False'} : Int;
   //    si16_CycleWriteAct { ExternalAccessible := 'False'; ExternalVisible := 'False'; ExternalWritable := 'False'} : Int;
   //    sbo_Write { ExternalAccessible := 'False'; ExternalVisible := 'False'; ExternalWritable := 'False'} : Bool;
   //    sbo_WriteEnergy { ExternalAccessible := 'False'; ExternalVisible := 'False'; ExternalWritable := 'False'} : Bool;
   //    sbo_WritePower { ExternalAccessible := 'False'; ExternalVisible := 'False'; ExternalWritable := 'False'} : Bool;
   //    sbo_WriteEnergyCounter { ExternalAccessible := 'False'; ExternalVisible := 'False'; ExternalWritable := 'False'} : Bool;
   //    sbo_WriteEnergyBusy { ExternalAccessible := 'False'; ExternalVisible := 'False'; ExternalWritable := 'False'} : Bool;
   //    sbo_WritePowerBusy { ExternalAccessible := 'False'; ExternalVisible := 'False'; ExternalWritable := 'False'} : Bool;
   //    sbo_WriteEnergyCounterBusy { ExternalAccessible := 'False'; ExternalVisible := 'False'; ExternalWritable := 'False'} : Bool;
   //    sbo_SyncPulseOld { ExternalAccessible := 'False'; ExternalVisible := 'False'; ExternalWritable := 'False'} : Bool;
   //    sbo_Alarm1 { ExternalAccessible := 'False'; ExternalVisible := 'False'; ExternalWritable := 'False'} : Bool;
   //    sbo_Alarm2 { ExternalAccessible := 'False'; ExternalVisible := 'False'; ExternalWritable := 'False'} : Bool;
   //    sbo_Alarm3 { ExternalAccessible := 'False'; ExternalVisible := 'False'; ExternalWritable := 'False'} : Bool;
   //    sbo_Alarm1Old { ExternalAccessible := 'False'; ExternalVisible := 'False'; ExternalWritable := 'False'} : Bool;
   //    sbo_Alarm2Old { ExternalAccessible := 'False'; ExternalVisible := 'False'; ExternalWritable := 'False'} : Bool;
   //    sbo_Alarm3Old { ExternalAccessible := 'False'; ExternalVisible := 'False'; ExternalWritable := 'False'} : Bool;
   //    sbo_ErrorAlarmState1 { ExternalAccessible := 'False'; ExternalVisible := 'False'; ExternalWritable := 'False'} : Bool;
   //    sbo_ErrorAlarmState2 { ExternalAccessible := 'False'; ExternalVisible := 'False'; ExternalWritable := 'False'} : Bool;
   //    sbo_ErrorAlarmState3 { ExternalAccessible := 'False'; ExternalVisible := 'False'; ExternalWritable := 'False'} : Bool;
   //    sbo_Init { ExternalAccessible := 'False'; ExternalVisible := 'False'; ExternalWritable := 'False'} : Bool;
   //    sb16_StatusAlarmState1 { ExternalAccessible := 'False'; ExternalVisible := 'False'; ExternalWritable := 'False'} : Word;
   //    sb16_StatusAlarmState2 { ExternalAccessible := 'False'; ExternalVisible := 'False'; ExternalWritable := 'False'} : Word;
   //    sb16_StatusAlarmState3 { ExternalAccessible := 'False'; ExternalVisible := 'False'; ExternalWritable := 'False'} : Word;
   // END_VAR
BEGIN
   energyMeta."name" := 'InfeedPAC3200';
   energyMeta.id[0] := 345;
   energyMeta.id[1] := 346;
   energyMeta.id[2] := 347;
   energyMeta.id[3] := 348;
   energyMeta.id[4] := 349;
   energyMeta.inputType := 2;
   energyMeta.configType := 2;
   energyMeta.mode := 1;
   energyMeta.syncPeriod := 60.0;
   energyMeta.overflowCntValue := 1000000.0;
   energyMeta.normFactorIn := 1.0;
   energyMeta.normFactorOut := 0.001;
   energyMeta.zeroCut := 0.0;
   energyMeta.baseAcqTime := 10.0;
   energyMeta.addAcqTime := 0.0;
   energyMeta.coordinationEnable := TRUE;
   energyMeta.cyclicRd := TRUE;
   energyMeta.cyclicTime := 10.0;
   energyMeta.unitActEnergy := 1179;
   energyMeta.unitActPower := 1190;
   energyMeta.unitAppEnergy := 1655;
   energyMeta.unitAppPower := 1652;
   energyMeta.unitReactEnergy := 1649;
   energyMeta.unitReactPower := 1646;
   energyMeta.unitPowerFactor := 1997;
   energyMeta.unitCurrent := 1209;
   energyMeta.unitVoltage := 1240;
   energyMeta.unitFrequency := 1077;
   energyMeta.unitAmpUnbalCurrent := 1342;
   energyMeta.unitAmpUnbalVoltage := 1342;
   energyMeta.archiveEnergy := TRUE;
   energyMeta.archivePower := TRUE;
   energyMeta.archiveEnergyCounter := TRUE;
END_DATA_BLOCK

DATA_BLOCK "InfeedPAC3200_Adv"   // DB36
TITLE = Instance DB of advanced energy data collection
// Instance DB of advanced energy data collection
// stored: InstanceOfName EnS_EnergyDataAdv, InstanceOfType FB
"EnS_EnergyDataAdv"
   // VAR_INPUT
   //    advData { ExternalWritable := 'False'} : "EnS_typeEnergyAdv";
   // END_VAR
   // VAR_OUTPUT
   //    error { ExternalAccessible := 'False'; ExternalVisible := 'False'; ExternalWritable := 'False'} : Bool;
   //    status { ExternalAccessible := 'False'; ExternalVisible := 'False'; ExternalWritable := 'False'} : Word;
   // END_VAR
   // VAR_IN_OUT
   //    orgData : "EnS_typeOrgData";
   //    energyMeta : "EnS_typeEnergyMeta";
   // END_VAR
BEGIN
END_DATA_BLOCK

DATA_BLOCK "InfeedPAC3200_AdvMinMax"   // DB37
TITLE = Instance DB of advanced min / max energy data collection
// Instance DB of advanced min / max energy data collection
// stored: InstanceOfName EnS_EnergyDataAdvMinMax, InstanceOfType FB
"EnS_EnergyDataAdvMinMax"
   // VAR_INPUT
   //    advDataMin { ExternalWritable := 'False'} : "EnS_typeEnergyAdv";
   //    advDataMax { ExternalWritable := 'False'} : "EnS_typeEnergyAdv";
   // END_VAR
   // VAR_OUTPUT
   //    error { ExternalAccessible := 'False'; ExternalVisible := 'False'; ExternalWritable := 'False'} : Bool;
   //    status { ExternalAccessible := 'False'; ExternalVisible := 'False'; ExternalWritable := 'False'} : Word;
   // END_VAR
BEGIN
END_DATA_BLOCK

DATA_BLOCK "EnS_Archive32469"   // DB8
TITLE = Instance DB of archiving function
// Instance DB of archiving function
// stored: InstanceOfName EnS_ArchiveHMI, InstanceOfType FB
"EnS_ArchiveHMI"
   // VAR_INPUT
   //    statusWrite : "EnS_typeHMIWriteStat";
   //    monitoringTime { ExternalAccessible := 'False'; ExternalVisible := 'False'; ExternalWritable := 'False'} : Time := T#30S;
   //    monitoringTimeWatchdog { ExternalAccessible := 'False'; ExternalVisible := 'False'; ExternalWritable := 'False'} : Time := T#5S;
   //    waitTime { ExternalAccessible := 'False'; ExternalVisible := 'False'; ExternalWritable := 'False'} : Time := T#1M;
   //    sD : Variant;
   //    messageSuppress { ExternalAccessible := 'False'; ExternalVisible := 'False'; ExternalWritable := 'False'} : Bool;
   // END_VAR
   // VAR_OUTPUT
   //    request : "EnS_typeHMIWriteCtrl";
   //    busy { ExternalAccessible := 'False'; ExternalVisible := 'False'; ExternalWritable := 'False'} : Bool;
   //    done { ExternalAccessible := 'False'; ExternalVisible := 'False'; ExternalWritable := 'False'} : Bool;
   //    error { ExternalAccessible := 'False'; ExternalVisible := 'False'; ExternalWritable := 'False'} : Bool;
   //    errorAlarm1 { ExternalAccessible := 'False'; ExternalVisible := 'False'; ExternalWritable := 'False'} : Bool;
   //    errorAlarm2 { ExternalAccessible := 'False'; ExternalVisible := 'False'; ExternalWritable := 'False'} : Bool;
   //    errorAlarm3 { ExternalAccessible := 'False'; ExternalVisible := 'False'; ExternalWritable := 'False'} : Bool;
   //    alarmState1 { ExternalAccessible := 'False'; ExternalVisible := 'False'; ExternalWritable := 'False'} : Byte;
   //    alarmState2 { ExternalAccessible := 'False'; ExternalVisible := 'False'; ExternalWritable := 'False'} : Byte;
   //    alarmState3 { ExternalAccessible := 'False'; ExternalVisible := 'False'; ExternalWritable := 'False'} : Byte;
   //    status { ExternalAccessible := 'False'; ExternalVisible := 'False'; ExternalWritable := 'False'} : Word;
   //    statusHMI { ExternalAccessible := 'False'; ExternalVisible := 'False'; ExternalWritable := 'False'} : Word;
   //    statusAlarm1 { ExternalAccessible := 'False'; ExternalVisible := 'False'; ExternalWritable := 'False'} : Word;
   //    statusAlarm2 { ExternalAccessible := 'False'; ExternalVisible := 'False'; ExternalWritable := 'False'} : Word;
   //    statusAlarm3 { ExternalAccessible := 'False'; ExternalVisible := 'False'; ExternalWritable := 'False'} : Word;
   // END_VAR
   // VAR_IN_OUT
   //    orgData : "EnS_typeOrgData";
   //    bufferWork : "EnS_typeBufferWork";
   // END_VAR
   // VAR
   //    Program_Alarm1 { ExternalAccessible := 'False'; ExternalVisible := 'False'; ExternalWritable := 'False'; S7_SetPoint := 'True'} : Program_Alarm;
   //    Program_Alarm2 { ExternalAccessible := 'False'; ExternalVisible := 'False'; ExternalWritable := 'False'; S7_SetPoint := 'True'} : Program_Alarm;
   //    Program_Alarm3 { ExternalAccessible := 'False'; ExternalVisible := 'False'; ExternalWritable := 'False'; S7_SetPoint := 'True'} : Program_Alarm;
   //    sbo_Req { ExternalAccessible := 'False'; ExternalVisible := 'False'; ExternalWritable := 'False'} : Bool;
   //    sbo_Repeat { ExternalAccessible := 'False'; ExternalVisible := 'False'; ExternalWritable := 'False'} : Bool;
   //    sbo_Wait { ExternalAccessible := 'False'; ExternalVisible := 'False'; ExternalWritable := 'False'} : Bool;
   //    sbo_Alarm1 { ExternalAccessible := 'False'; ExternalVisible := 'False'; ExternalWritable := 'False'} : Bool;
   //    sbo_Alarm2 { ExternalAccessible := 'False'; ExternalVisible := 'False'; ExternalWritable := 'False'} : Bool;
   //    sbo_Alarm3 { ExternalAccessible := 'False'; ExternalVisible := 'False'; ExternalWritable := 'False'} : Bool;
   //    sbo_Alarm1Old { ExternalAccessible := 'False'; ExternalVisible := 'False'; ExternalWritable := 'False'} : Bool;
   //    sbo_Alarm2Old { ExternalAccessible := 'False'; ExternalVisible := 'False'; ExternalWritable := 'False'} : Bool;
   //    sbo_Alarm3Old { ExternalAccessible := 'False'; ExternalVisible := 'False'; ExternalWritable := 'False'} : Bool;
   //    sbo_ErrorAlarmState1 { ExternalAccessible := 'False'; ExternalVisible := 'False'; ExternalWritable := 'False'} : Bool;
   //    sbo_ErrorAlarmState2 { ExternalAccessible := 'False'; ExternalVisible := 'False'; ExternalWritable := 'False'} : Bool;
   //    sbo_ErrorAlarmState3 { ExternalAccessible := 'False'; ExternalVisible := 'False'; ExternalWritable := 'False'} : Bool;
   //    sbo_Init { ExternalAccessible := 'False'; ExternalVisible := 'False'; ExternalWritable := 'False'} : Bool;
   //    su32_NoItems { ExternalAccessible := 'False'; ExternalVisible := 'False'; ExternalWritable := 'False'} : UDInt;
   //    su32_NoDeletedItems { ExternalAccessible := 'False'; ExternalVisible := 'False'; ExternalWritable := 'False'} : UDInt;
   //    si32_WriteHMIItem { ExternalAccessible := 'False'; ExternalVisible := 'False'; ExternalWritable := 'False'} : UDInt;
   //    sb16_StatusArchiving { ExternalAccessible := 'False'; ExternalVisible := 'False'; ExternalWritable := 'False'} : Word;
   //    su16_MonitoringTime { ExternalAccessible := 'False'; ExternalVisible := 'False'; ExternalWritable := 'False'} : UInt;
   //    su16_MonitoringTimeWatchdog { ExternalAccessible := 'False'; ExternalVisible := 'False'; ExternalWritable := 'False'} : UInt;
   //    su16_WaitTime { ExternalAccessible := 'False'; ExternalVisible := 'False'; ExternalWritable := 'False'} : UInt;
   //    sb16_StatusAlarmState1 { ExternalAccessible := 'False'; ExternalVisible := 'False'; ExternalWritable := 'False'} : Word;
   //    sb16_StatusAlarmState2 { ExternalAccessible := 'False'; ExternalVisible := 'False'; ExternalWritable := 'False'} : Word;
   //    sb16_StatusAlarmState3 { ExternalAccessible := 'False'; ExternalVisible := 'False'; ExternalWritable := 'False'} : Word;
   //    sldt_TimeStamp { ExternalAccessible := 'False'; ExternalVisible := 'False'; ExternalWritable := 'False'} : LDT;
   // END_VAR
BEGIN
END_DATA_BLOCK

